	FOR NB2 := 1 TO NB_GROUP DO
		IF TBL_GROUP[NB2].NOM	= '' THEN
			IF NB2 < NB_GROUP THEN
				IF TBL_GROUP[NB2+1].NOM	<> '' THEN
					TBL_GROUP[NB2].NOM				:=	TBL_GROUP[NB2+1].NOM;
					TBL_GROUP[NB2].CONF_MACHINE	:=	TBL_GROUP[NB2+1].CONF_MACHINE;
					TBL_GROUP[NB2].FONCTION_SA		:=	TBL_GROUP[NB2+1].FONCTION_SA;
					TBL_GROUP[NB2].MAINTENANCE		:=	TBL_GROUP[NB2+1].MAINTENANCE;
					TBL_GROUP[NB2].PRODUCTION		:=	TBL_GROUP[NB2+1].PRODUCTION;
					TBL_GROUP[NB2].PROGRAMMATION	:=	TBL_GROUP[NB2+1].PROGRAMMATION;
					TBL_GROUP[NB2].SUPERVISEUR		:=	TBL_GROUP[NB2+1].SUPERVISEUR;
					TBL_GROUP[NB2].CONF_TRF			:=	TBL_GROUP[NB2+1].CONF_TRF;
					TBL_GROUP[NB2].MODIF_ENLIGNE	:=	TBL_GROUP[NB2+1].MODIF_ENLIGNE;
					TBL_GROUP[NB2].ARCHIVE_EV		:=	TBL_GROUP[NB2+1].ARCHIVE_EV;
					TBL_GROUP[NB2].DECONSIGNATION	:=	TBL_GROUP[NB2+1].DECONSIGNATION;
					TBL_GROUP[NB2+1].NOM				:=	'';
					TBL_GROUP[NB2+1].CONF_MACHINE	:=	FALSE;
					TBL_GROUP[NB2+1].FONCTION_SA	:=	FALSE;
					TBL_GROUP[NB2+1].MAINTENANCE	:=	FALSE;
					TBL_GROUP[NB2+1].PRODUCTION		:=	FALSE;
					TBL_GROUP[NB2+1].PROGRAMMATION	:=	FALSE;
					TBL_GROUP[NB2+1].SUPERVISEUR		:=	FALSE;
					TBL_GROUP[NB2+1].CONF_TRF			:=	FALSE;
					TBL_GROUP[NB2+1].MODIF_ENLIGNE		:=	FALSE;
					TBL_GROUP[NB2+1].ARCHIVE_EV			:=	FALSE;
					TBL_GROUP[NB2+1].DECONSIGNATION	:=	FALSE;
				END_IF
			END_IF
		END_IF;
	END_FOR;

	DD_ORG_GRP	:=	FALSE;
END_IF
(*================================================================================================*)


(****************************************************** 	Organisation des utlisateurs après suppression **********************************************)
IF DD_ORG_USER THEN
	FOR NB := 1 TO NB_USER DO
		IF  TBL_USER[NB].LOGIN = '' THEN
			IF NB < NB_USER THEN
				IF  TBL_USER[NB+1].LOGIN <> '' THEN
					TBL_USER[NB].LOGIN		:=	TBL_USER[NB+1].LOGIN;
					TBL_USER[NB].GROUPE	:=	TBL_USER[NB+1].GROUPE;
					TBL_USER[NB].NOM		:=	TBL_USER[NB+1].NOM;
					TBL_USER[NB].PRENOM	:=	TBL_USER[NB+1].PRENOM;
					TBL_USER[NB].PASS		:=	TBL_USER[NB+1].PASS;
					TBL_USER[NB+1].LOGIN		:=	'';
					TBL_USER[NB+1].GROUPE		:=	'';
					TBL_USER[NB+1].NOM			:=	'';
					TBL_USER[NB+1].PRENOM	:=	'';
					TBL_USER[NB+1].PASS		:=	'';
				END_IF
			END_IF
		END_IF
	END_FOR

	DD_ORG_USER	:=	FALSE;
END_IF
(*================================================================================================*)



(****************************************************** 	Autorisation modification nom du groupe ***************************************************)
TROUV:=FALSE;
FOR NB := 1 TO NB_GROUP DO
	IF nb <> LIGNE_GROUP THEN
		IF TBL_GROUP[NB].NOM = GROUP_TEMP.NOM THEN
			TROUV := TRUE;
		END_IF
	END_IF
END_FOR
FOR NB := 1 TO NB_USER DO
	IF TBL_USER[NB].GROUPE = TBL_GROUP[LIGNE_GROUP].NOM AND TBL_GROUP[LIGNE_GROUP].NOM <> GROUP_TEMP.NOM THEN
		TROUV		:=	TRUE;
	END_IF
END_FOR
IF TROUV THEN
	AUT_NOM_GRP	:=	FALSE;
ELSE
	AUT_NOM_GRP	:=	TRUE;
END_IF
(*================================================================================================*)



(****************************************************** 	Autorisation modification nom des utilisateurs ***************************************************)
TROUV:=FALSE;
FOR NB := 1 TO NB_USER DO
	IF nb <> LIGNE THEN
		IF TBL_USER[NB].LOGIN = USER_TEMP.LOGIN THEN
			TROUV := TRUE;
		END_IF
	END_IF
END_FOR
IF TROUV THEN
	AUT_NOM_USER	:=	FALSE;
ELSE
	AUT_NOM_USER	:=	TRUE;
END_IF
(*================================================================================================*)



(****************************************************** 	Autorisation création utilisateur ***************************************************)
IF USER_TEMP.LOGIN = '' OR USER_TEMP.PASS = '' OR USER_TEMP.PASS <> PASS_CONF OR USER_TEMP.LOGIN = 'ac' THEN
	AUT_NEW_USER	:=	FALSE;
ELSE
	AUT_NEW_USER	:=	TRUE;
END_IF
(*================================================================================================*)


(********************************************************** Gestion du logout automatique **************************************************)
IF OPT_LOGOUT THEN
	TPS_ECOUL.IN		:=	UTIL_EC AND NOT MANUFACTURER;
	TPS_ECOUL.PT	:=	TIM_LOGOUT;
	TPS_ECOUL();
	IF TPS_ECOUL.Q AND NOT MACHINE.STATE_Prod THEN
		DD_DELOG	:=	TRUE;
	END_IF
END_IF
(*=========================================================================================*)

(********************************************************** Autorisation utilisation logout auto **************************************************)
IF TIM_LOGOUT > T#10s THEN
	AUT_OPT_LOGOUT	:=	TRUE;
ELSE
	AUT_OPT_LOGOUT	:=	FALSE;
END_IF
(*=========================================================================================*)

END_FUNCTION_BLOCK

// ---- POUs/Programme/BLOCK_PRG_EFFLUVAGE.TcPOU
FUNCTION_BLOCK BLOCK_PRG_EFFLUVAGE
VAR
END_VAR
VAR_INPUT PERSISTENT
(* Entité*)
	IsAssembly:			 	BOOL;					(*entité de type fonction*)
	TagXml:					UINT;
	IdXml: 					STRING;
	IdParent: 				STRING;					(*MNEMO du pére*)
	MNEMO:					STRING;					(*MNEMO de cette entité *)
END_VAR
VAR_INPUT
END_VAR
VAR_OUTPUT
	STATE_AR:				BOOL;
	STATE_Def_IProc:		BOOL;		(*I_STANDARD -indique la présence d'un défaut entrainant l'arrêt du procédé*)
END_VAR

(* Parametre statique *)
(*General*)
IdParent			:= 	'';
MNEMO				:=	'EFFLUV';
IdXML				:=	'15';
TagXML				:=	0;


STATE_AR := TRUE;
STATE_Def_IProc := FALSE;

END_FUNCTION_BLOCK

// ---- POUs/Programme/BLOCK_PRG_EVAP.TcPOU
FUNCTION_BLOCK BLOCK_PRG_EVAP
VAR_INPUT
(*Quartz*)
	QZ1:				BLOCK_XTAL6; 	(*Tête Quartz*)
	XTC3:				BLOCK_XTC3;	(*Contrôleur de dépôt XTC3*)

(*Evenement*)
	EV_SHUTTER1_OPEN:	PRCDEF;		(*Evenement cache source 1 ouvert*)
	EV_SHUTTER1_CLOSE:	PRCDEF;		(*Evenement cache source 1 fermé*)

	EV_SHUTTER2_OPEN:	PRCDEF;		(*Evenement cache source 2 ouvert*)
	EV_SHUTTER2_CLOSE:	PRCDEF;		(*Evenement cache source 2 fermé*)

	EV_SHUTTER3_OPEN:	PRCDEF;		(*Evenement cache source 3 ouvert*)
	EV_SHUTTER3_CLOSE:	PRCDEF;		(*Evenement cache source 3 fermé*)

(*Entrées*)
	(*Creuset*)
	IN_CR11T		AT%I*:		BOOL;		(*Creuset en position 1*)
	IN_CR12T		AT%I*:		BOOL;		(*Creuset en position 2*)
	IN_CR13T		AT%I*:		BOOL;		(*Creuset en position 3*)
	IN_CR14T		AT%I*:		BOOL;		(*Creuset en position 4*)

	(*Balayage*)
	IN_SW_REM		AT%I*:		BOOL;		(*Balayage en mode remote*)
	IN_SW_RUN		AT%I*:		BOOL;		(*Balayage en marche*)
	IN_SW_RDY		AT%I*:		BOOL;		(*Balayage prêt*)

	VISU_STOP_ECO_MANU:			BOOL;
END_VAR
VAR_INPUT PERSISTENT
	(*Entité*)
	IsAssembly:		BOOL;			(*entité : ensemble*)
	IdXML:			STRING;			(*nom entité : identifiant pour recherche dans dico*)
	TagXML:			UINT;			(*nom entité : identifiant pour recherche dans dico*)
	IdParent:		STRING;			(*MNEMO de l'appelant*)
	MNEMO:			STRING;			(*MNEMO de l'entité*)

	CONF_QUARTZ_CC_SRCE:	ARRAY[0..4] OF BOOL;	(*Indique si un Quartz se trouve sous le cache source pour contrôle vitesse pendant phase de préfusion*)
	CONF_CHAUFFAGE:			BOOL; 	(*Indique s'il y a du chauffage*)
	CONF_IAD:				BOOL;	(*Indique s'il y a un IAD*)

	PRM_Seuil_Crystal_Life:			REAL;	(*Seuil d'alarme pour la vie des quartz*)
	PRM_Seuil_Crystal_Activity:		REAL;	(*Seuil d'alarme pour l'activité des quartz*)

	PRM_Forcage_Crucible:		BOOL;	(*Option de forçage du creuset en semi-auto*)
	PRM_Forcage_Cache_Source1:	BOOL;	(*Option de forçage du cache source 1 en semi-auto*)
	PRM_Forcage_Cache_Source2:	BOOL;	(*Option de forçage du cache source 2 en semi-auto*)
	PRM_Forcage_Cache_Source3:	BOOL;	(*Option de forçage du cache source 3 en semi-auto*)
	PRM_Forcage_Cache_Quartz:	BOOL;	(*Option de forçage du cache quartz en semi-auto*)

	PRM_Adresse_IP_XTC:			STRING(15) := '192.168.0.20'; (*Addresse IP de l'XTC affecté depuis l'IHM*)

	PRM_Mat_Source2:			STRING; (*Nom du matériau utilisé sur la source 2*)
	PRM_Mat_Source3:			STRING; (*Nom du matériau utilisé sur la source 3*)
END_VAR

VAR
	EVAPS1:			BLOCK_EVAP;
	EVAPS2:			BLOCK_EVAP;
	EVAPS3:			BLOCK_EVAP;
	CC11:			BLOCK_ACTUATOR;
	CC12:			BLOCK_ACTUATOR;
	CC13:			BLOCK_ACTUATOR;
	SOURCE1:		BLOCK_CANON_ST10;
	SOURCE2:		BLOCK_SOURCE_JOULE;
	SOURCE3:		BLOCK_SOURCE_JOULE;
	SWEEP1:			BLOCK_TELEMARK_CHEETAH_SWEEP;
	CRUCIBLE1:		BLOCK_IND_CR_396_TELEMARK;

	VAR_Idx:		INT;				(*Variable d'itération*)

	(*Variable Bidon*)
	VAR_NCR:				USINT;
	VAR_NBAL:				USINT;
	VAR_HT:					REAL;
END_VAR

VAR_OUTPUT
	STATE_AR:						BOOL;
	STATE_Def_IProc:   				BOOL;		(*Etat de défaut*)
	(*Caches*)
	OUT_OCC11			AT%Q*:		BOOL;		(*Ouverture cache source 1*)
	OUT_ICC11			AT%Q*:		BOOL;		(*Fermeture cache source 1*)
	OUT_OCC12			AT%Q*:		BOOL;		(*Ouverture cache source 2*)
	OUT_ICC12			AT%Q*:		BOOL;		(*Fermeture cache source 2*)
	OUT_OCC13			AT%Q*:		BOOL;		(*Ouverture cache source 3*)
	OUT_ICC13			AT%Q*:		BOOL;		(*Fermeture cache source 3*)
	(*Creuset*)
	OUT_CR11			AT%Q*:		BOOL;		(*Sélection du creuset 1*)
	OUT_CR12			AT%Q*:		BOOL;		(*Sélection du creuset 2*)
	OUT_CR13			AT%Q*:		BOOL;		(*Sélection du creuset 3*)
	OUT_CR14			AT%Q*:		BOOL;		(*Sélection du creuset 4*)
	OUT_CR_RMT			AT%Q*:		BOOL;		(*remote indexeur de creuset*)
	(*Sweep*)
	OUT_SWB1			AT%Q*:		BOOL;		(*Sélection programme de balayage bit 1*)
	OUT_SWB2			AT%Q*:		BOOL;		(*Sélection programme de balayage bit 2*)
	OUT_SWB3			AT%Q*:		BOOL;		(*Sélection programme de balayage bit 3*)
	OUT_SWB4			AT%Q*:		BOOL;		(*Sélection programme de balayage bit 4*)
	//OUT_SWITLK			AT%Q*:		BOOL;		(*Interlock module balayage*)
	OUT_SWP_ON			AT%Q*:		BOOL;		(*activation balayage*)
	OUT_SW_RMT			AT%Q*:		BOOL;		(*remote module de balayage*)
	(*Effet joule*)
	OUT_MEJ1			AT%Q*:		BOOL;
	OUT_MEJ2			AT%Q*:		BOOL;
	OUT_QEJ1			AT%Q*:		INT;
	OUT_QEJ2			AT%Q*:		INT;
	
	(*Divers*)
	OUT_MEG1			AT%Q*:		BOOL;		(*Sécurité vide canon pour mise en puissance canons + ECO-MODE*)
	OUT_MPR230			AT%Q*:		BOOL;		(*230V Module Balayage + Module Indexage + XTC ECO-MODE*)
	ECO_MODE:						BOOL;

	O_END_PROCESS_PFIXE:			BOOL;		(**)
END_VAR

VAR
	TIMER_ECO_MODE:					TOF;
END_VAR

(*General*)
IdParent					:=	MACHINE.MNEMO;
MNEMO						:=	CONCAT(IdParent,'_EVAP');
IdXML						:=	'17';
TagXML						:=	0;

(*XTC3*)
XTC3.MNEMO					:=	'XTC3';
XTC3.IdXML					:=	'19';
XTC3.TagXML					:=	1;

(*Quartz*)
QZ1.MNEMO					:=	'QZ1';
QZ1.IdParent				:=	MNEMO;

(*Source1*)
SOURCE1.IdParent			:=	MNEMO;
SOURCE1.MNEMO				:=	'Canon e-';
SOURCE1.IdXML				:=	'16';
SOURCE1.TagXML 				:= 	3;

(*Source2*)
SOURCE2.IdParent			:=	MNEMO;
SOURCE2.MNEMO				:=	'Source J-Gauche';
SOURCE2.IdXML				:=	'16';
SOURCE2.TagXML				:=	4;

(*Source3*)
SOURCE3.IdParent			:=	MNEMO;
SOURCE3.MNEMO				:=	'Source J-Droite';
SOURCE3.IdXML				:=	'16';
SOURCE3.TagXML				:=	5;

(*Balayage*)
SWEEP1.IdParent				:=	SOURCE1.MNEMO;
SWEEP1.MNEMO				:=	'SWP1';
SWEEP1.IdXML				:=	'16';
SWEEP1.TagXML				:=	8;

(*Indexeur*)
CRUCIBLE1.IdParent 			:=	SOURCE1.MNEMO;
CRUCIBLE1.MNEMO 			:=	'INDCR1';
CRUCIBLE1.IdXML				:=	'16';
CRUCIBLE1.TagXML 			:=  7;

CRUCIBLE1.CONF_NCR			:= 	4;			(*Nombre de creuset de l'indexeur*)

(*Cache CC11*)
CC11.CONF_Tim_Valid_Off			:=	T#0ms;
CC11.CONF_Tim_Valid_On			:=	T#0ms;
CC11.DEF_Off.DELAY				:=	T#10s;
CC11.DEF_On.DELAY				:=	T#10s;
CC11.DEF_Sensor.DELAY			:=	T#10s;
CC11.CONF_DI_Off				:=	FALSE;
CC11.CONF_DI_On					:=	FALSE;
CC11.CONF_No_Safety_Auto		:=	TRUE;
CC11.CONF_Type_Actuator			:=	0;
CC11.MNEMO						:=	'Canon e-';
CC11.CONF_EN_On					:=	0;
CC11.CONF_No_Safety_Auto		:=	FALSE;
CC11.IdXML						:=	'4';
CC11.TagXML						:=	1;
CC11.IdParent					:=	Source1.MNEMO;
CC11.DEF_Off_auto.IdXML			:=	'3';
CC11.DEF_Off_auto.TagXML		:=	11;
CC11.DEF_Off_Imposs.IdXML		:=	'3';
CC11.DEF_Off_Imposs.TagXML		:=	9;
CC11.DEF_On_Imposs.IdXML		:=	'3';
CC11.DEF_On_Imposs.TagXML		:=	6;
CC11.DEF_Off.IdXML				:=	'3';
CC11.DEF_Off.TagXML 			:=	4;
CC11.DEF_On.IdXML				:=	'3';
CC11.DEF_On.TagXML 				:=	2;
CC11.DEF_Sensor.IdXML			:=	'3';
CC11.DEF_Sensor.TagXML 			:=	13;

(*Cache CC12*)
CC12.CONF_Tim_Valid_Off			:=	T#0ms;
CC12.CONF_Tim_Valid_On			:=	T#0ms;
CC12.DEF_Off.DELAY				:=	T#10s;
CC12.DEF_On.DELAY				:=	T#10s;
CC12.DEF_Sensor.DELAY			:=	T#10s;
CC12.CONF_DI_Off				:=	FALSE;
CC12.CONF_DI_On					:=	FALSE;
CC12.CONF_No_Safety_Auto		:=	TRUE;
CC12.CONF_Type_Actuator			:=	0;
CC12.MNEMO						:=	'SJ-Gauche';
CC12.CONF_EN_On					:=	0;
CC12.CONF_No_Safety_Auto		:=	FALSE;
CC12.IdXML						:=	'4';
CC12.TagXML						:=	1;
CC12.IdParent					:=	Source2.MNEMO;
CC12.DEF_Off_auto.IdXML			:=	'3';
CC12.DEF_Off_auto.TagXML		:=	11;
CC12.DEF_Off_Imposs.IdXML		:=	'3';
CC12.DEF_Off_Imposs.TagXML		:=	9;
CC12.DEF_On_Imposs.IdXML		:=	'3';
CC12.DEF_On_Imposs.TagXML		:=	6;
CC12.DEF_Off.IdXML				:=	'3';
CC12.DEF_Off.TagXML 			:=	4;
CC12.DEF_On.IdXML				:=	'3';
CC12.DEF_On.TagXML 				:=	2;
CC12.DEF_Sensor.IdXML			:=	'3';
CC12.DEF_Sensor.TagXML 			:=	13;

(*Cache CC13*)
CC13.CONF_Tim_Valid_Off			:=	T#0ms;
CC13.CONF_Tim_Valid_On			:=	T#0ms;
CC13.DEF_Off.DELAY				:=	T#10s;
CC13.DEF_On.DELAY				:=	T#10s;
CC13.DEF_Sensor.DELAY			:=	T#10s;
CC13.CONF_DI_Off				:=	FALSE;
CC13.CONF_DI_On					:=	FALSE;
CC13.CONF_No_Safety_Auto		:=	TRUE;
CC13.CONF_Type_Actuator			:=	0;
CC13.MNEMO						:=	'SJ-Droite';
CC13.CONF_EN_On					:=	0;
CC13.CONF_No_Safety_Auto		:=	FALSE;
CC13.IdXML						:=	'4';
CC13.TagXML						:=	1;
CC13.IdParent					:=	Source3.MNEMO;
CC13.DEF_Off_auto.IdXML			:=	'3';
CC13.DEF_Off_auto.TagXML		:=	11;
CC13.DEF_Off_Imposs.IdXML		:=	'3';
CC13.DEF_Off_Imposs.TagXML		:=	9;
CC13.DEF_On_Imposs.IdXML		:=	'3';
CC13.DEF_On_Imposs.TagXML		:=	6;
CC13.DEF_Off.IdXML				:=	'3';
CC13.DEF_Off.TagXML 			:=	4;
CC13.DEF_On.IdXML				:=	'3';
CC13.DEF_On.TagXML 				:=	2;
CC13.DEF_Sensor.IdXML			:=	'3';
CC13.DEF_Sensor.TagXML 			:=	13;

EVAPS1.IdXML 				:=	'17';
EVAPS1.TagXML				:=	1;
EVAPS1.CONF_No_Sweep		:=	FALSE;
EVAPS1.DEF_Pmax.DELAY		:=	T#10S;
EVAPS1.DEF_Pmin.DELAY		:=	T#10s;

EVAPS2.IdXML				:=	'17';
EVAPS2.TagXML				:=	2;
EVAPS2.CONF_No_Sweep		:=	TRUE;
EVAPS2.DEF_Pmax.DELAY		:=	T#10S;
EVAPS2.DEF_Pmin.DELAY		:=	T#10s;

EVAPS3.IdXML				:=	'17';
EVAPS3.TagXML				:=	3;
EVAPS3.CONF_No_Sweep		:=	TRUE;
EVAPS3.DEF_Pmax.DELAY		:=	T#10S;
EVAPS3.DEF_Pmin.DELAY		:=	T#10s;


EV_SHUTTER1_OPEN.IdXML			:=	'14';
EV_SHUTTER1_OPEN.TagXML			:=	20;
EV_SHUTTER1_OPEN.Groupe			:=	3;

EV_SHUTTER1_CLOSE.IdXML			:=	'14';
EV_SHUTTER1_CLOSE.TagXML		:=	21;
EV_SHUTTER1_CLOSE.Groupe		:=	3;

EV_SHUTTER2_OPEN.IdXML			:=	'14';
EV_SHUTTER2_OPEN.TagXML			:=	24;
EV_SHUTTER2_OPEN.Groupe			:=	3;

EV_SHUTTER2_CLOSE.IdXML			:=	'14';
EV_SHUTTER2_CLOSE.TagXML		:=	25;
EV_SHUTTER2_CLOSE.Groupe		:=	3;

EV_SHUTTER3_OPEN.IdXML			:=	'14';
EV_SHUTTER3_OPEN.TagXML			:=	26;
EV_SHUTTER3_OPEN.Groupe			:=	3;

EV_SHUTTER3_CLOSE.IdXML			:=	'14';
EV_SHUTTER3_CLOSE.TagXML		:=	27;
EV_SHUTTER3_CLOSE.Groupe		:=	3;


CONF_CHAUFFAGE:= FALSE;
CONF_IAD:=FALSE;

CONF_QUARTZ_CC_SRCE[0]:= FALSE;
CONF_QUARTZ_CC_SRCE[1]:= FALSE;
CONF_QUARTZ_CC_SRCE[2]:= FALSE;
CONF_QUARTZ_CC_SRCE[3]:= FALSE;
CONF_QUARTZ_CC_SRCE[4]:= FALSE;


(*mode de controle des fonctions*)
IF MACHINE.RQ_Ctrl_Ihm THEN
	QZ1.CTRL_PLC := FALSE;
ELSIF MACHINE.RQ_Ctrl_Plc THEN
	QZ1.CTRL_PLC := TRUE;
END_IF

(*Configuration Adresse IP XTC*)
XTC3.CONF_sRemoteHost:= PRM_Adresse_IP_XTC;
XTC3.CONF_nRemotePort := 2101;


(*Evenement ouverture cache source 1*)
EV_SHUTTER1_OPEN.CONDITION	:= MACHINE.STATE_Prod AND CC11.STATE_On;
EV_SHUTTER1_OPEN();
(*Evenement fermeture cache source 1*)
EV_SHUTTER1_CLOSE.CONDITION:= MACHINE.STATE_Prod AND CC11.STATE_Off;
EV_SHUTTER1_CLOSE();

(*Evenement ouverture cache source 2*)
EV_SHUTTER2_OPEN.CONDITION	:= MACHINE.STATE_Prod AND CC12.STATE_On;
EV_SHUTTER2_OPEN();
(*Evenement fermeture cache source 2*)
EV_SHUTTER2_CLOSE.CONDITION:= MACHINE.STATE_Prod AND CC12.STATE_Off;
EV_SHUTTER2_CLOSE();

(*Evenement ouverture cache source 3*)
EV_SHUTTER3_OPEN.CONDITION	:= MACHINE.STATE_Prod AND CC13.STATE_On;
EV_SHUTTER3_OPEN();
(*Evenement fermeture cache source 3*)
EV_SHUTTER3_CLOSE.CONDITION:= MACHINE.STATE_Prod AND CC13.STATE_Off;
EV_SHUTTER3_CLOSE();


(*Reset des ordres de forçage*)
IF MACHINE.RQ_Start_Prod OR MACHINE.STATE_Off OR MACHINE.STATE_Manu THEN
	PRM_Forcage_Crucible 		:= 	FALSE;
	PRM_Forcage_Cache_Source1	:= 	FALSE;
	PRM_Forcage_Cache_Source2	:=	FALSE;
	PRM_Forcage_Cache_Source3  	:=	FALSE;
	PRM_Forcage_Cache_Quartz	:=	FALSE;
END_IF
IF CRUCIBLE1.DEF_POSITIONNEMENT.DEF THEN
	PRM_Forcage_Crucible		:= FALSE;
END_IF
IF CC11.DEF_Off_auto.DEF THEN
	PRM_Forcage_Cache_Source1:= FALSE;
END_IF
IF CC12.DEF_Off_auto.DEF	THEN
	PRM_Forcage_Cache_Source2:= FALSE;
END_IF
IF CC13.DEF_Off_auto.DEF	THEN
	PRM_Forcage_Cache_Source3:= FALSE;
END_IF


(******************* SOURCE 1 **********************)

SOURCE1.HV.EN_Off_EXT := TRUE;
SOURCE1.HV.EN_On_EXT := (SWEEP1.STATE_REM AND SWEEP1.STATE_ON);

SOURCE1(
	DOOR:= PRG_POMPAGE.DOOR,
	VAC:= (PRG_POMPAGE.VAC AND PRG_POMPAGE.M11.STATE_Seuil[13] AND NOT PRG_POMPAGE.POMPAGE.VS11.STATE_Off),
	WATER:= PRG_SERVITUDES.WATER[4] AND PRG_SERVITUDES.WATER[5],	(*Refroidissement canon à électrons*)
	MANUAL:= MACHINE.STATE_Manu,
	I_CR_OK:= CRUCIBLE1.STATE_POS_OK,
	RESET:= MACHINE.STATE_Off,
	I_COURANT:= EVAPS1.OUT_Power,
	CO_HV:= EVAPS1.RQ_marche_HT,
	CO_SRC:=EVAPS1.RQ_marche_FIL ,);

SWEEP1(
	MANUAL:= MACHINE.STATE_Manu,
	RESET:= MACHINE.STATE_Off,
	DOOR:= PRG_POMPAGE.DOOR,
	CO_Remote:= MACHINE.STATE_Auto,
	CO_balayage:= MACHINE.STATE_Auto AND EVAPS1.RQ_marche_SWEEP,
	I_SW_RUN:= IN_SW_RUN,
	I_SW_RDY:= IN_SW_RDY,
	OUT_SWB1 => OUT_SWB1,
	OUT_SWB2 => OUT_SWB2,
	OUT_SWB3 => OUT_SWB3,
	OUT_SWB4 => OUT_SWB4,
	OUT_SWP_ON => OUT_SWP_ON,
	OUT_RMT	=> OUT_SW_RMT);

CRUCIBLE1(
	MANUAL:= MACHINE.STATE_Manu,
	RESET:= MACHINE.STATE_Off,
	CO_Change:= EVAPS1.RQ_Switch_Crucible OR PRM_Forcage_Crucible,
	I_FIL_ON:= SOURCE1.STATE_SRC_ON,
	IN_POWER:= EVAPS1.OUT_Power,
	IN_POS1:= IN_CR11T,
	IN_POS2:= IN_CR12T,
	IN_POS3:= IN_CR13T,
	IN_POS4:= IN_CR14T,
	OUT_SEL1=> OUT_CR11,
	OUT_SEL2=> OUT_CR12,
	OUT_SEL3=> OUT_CR13,
	OUT_SEL4=> OUT_CR14);

CC11(
	RESET:= MACHINE.STATE_Off ,
	MANUAL:=MACHINE.STATE_Manu,
	IN_OFF:= ,
	IN_ON:= ,
	CO_On:= EVAPS1.RQ_Ouv_Cache_source OR PRM_Forcage_Cache_Source1,
	CO_Off:= NOT EVAPS1.RQ_Ouv_Cache_source AND NOT PRM_Forcage_Cache_Source1 AND NOT MACHINE.STATE_Manu AND NOT MACHINE.STATE_Off,
	EN_On_INT:= TRUE,
	EN_Off_INT:= TRUE,
	EN_On_EXT:=TRUE,
	EN_Off_EXT:= TRUE,
	OUT_On=> OUT_OCC11,
	OUT_Off=> OUT_ICC11,);
	

(******************* SOURCE 2 **********************)

SOURCE2.EJ.EN_Off_EXT	:=	TRUE;
SOURCE2.EJ.EN_On_EXT	:=	NOT SOURCE3.OUT_MEJ;

SOURCE2(
	DOOR:=					PRG_POMPAGE.DOOR,
	VAC:=					PRG_POMPAGE.VAC AND NOT PRG_POMPAGE.POMPAGE.VS11.STATE_Off,
	WATER:=					PRG_SERVITUDES.WATER[2],					(*Refroidissement Source Joule n°1*)
	MANUAL:=				MACHINE.STATE_Manu,
	I_CR_OK:=				TRUE,										(*Positionnement du creuset ok*)
	RESET:=					MACHINE.STATE_Off,
	I_POWER:=				EVAPS2.OUT_Power,
	CO_SRC:=				EVAPS2.RQ_marche_HT, );

CC12(
	RESET:= MACHINE.STATE_Off ,
	MANUAL:=MACHINE.STATE_Manu,
	IN_OFF:= ,
	IN_ON:= ,
	CO_On:= EVAPS2.RQ_Ouv_Cache_source OR PRM_Forcage_Cache_Source2,
	CO_Off:= NOT EVAPS2.RQ_Ouv_Cache_source AND NOT PRM_Forcage_Cache_Source2 AND NOT MACHINE.STATE_Manu AND NOT MACHINE.STATE_Off,
	EN_On_INT:= TRUE,
	EN_Off_INT:= TRUE,
	EN_On_EXT:=TRUE,
	EN_Off_EXT:= TRUE,
	OUT_On=> OUT_OCC12,
	OUT_Off=> OUT_ICC12);

(******************* SOURCE 3 **********************)

SOURCE3.EJ.EN_Off_EXT	:=	TRUE;
SOURCE3.EJ.EN_On_EXT	:=	NOT SOURCE2.OUT_MEJ;

SOURCE3(
	DOOR:=					PRG_POMPAGE.DOOR,
	VAC:=					PRG_POMPAGE.VAC AND NOT PRG_POMPAGE.POMPAGE.VS11.STATE_Off,
	WATER:=					PRG_SERVITUDES.WATER[3],					(*Refroidissement Source Joule n°2*)
	MANUAL:=				MACHINE.STATE_Manu,
	I_CR_OK:=				TRUE,										(*Positionnement du creuset ok*)
	RESET:=					MACHINE.STATE_Off,
	I_POWER:=				EVAPS3.OUT_Power,
	CO_SRC:=				EVAPS3.RQ_marche_HT,	);

	
CC13(
	RESET:= MACHINE.STATE_Off ,
	MANUAL:= MACHINE.STATE_Manu,
	IN_OFF:= ,
	IN_ON:= ,
	CO_On:= EVAPS3.RQ_Ouv_Cache_source OR PRM_Forcage_Cache_Source3,
	CO_Off:= NOT EVAPS3.RQ_Ouv_Cache_source AND NOT PRM_Forcage_Cache_Source3 AND NOT MACHINE.STATE_Manu AND NOT MACHINE.STATE_Off,
	EN_On_INT:= TRUE,
	EN_Off_INT:= TRUE,
	EN_On_EXT:=TRUE,
	EN_Off_EXT:= TRUE,
	OUT_On=> OUT_OCC13,
	OUT_Off=> OUT_ICC13,);
	
(******************* QUARTZ **********************)

(*Quartz QZ1*)
IF MACHINE.STATE_Prod THEN
	IF MAIN.STEP_EMPILEMENT.PRM_UTIL_SOURCE1 THEN
		QZ1.PRM_CONS_POSITION_QZ:= EVAPS1.OUT_Cons_Pos_Qz;
	END_IF
	IF MAIN.STEP_EMPILEMENT.PRM_UTIL_SOURCE2 THEN
		QZ1.PRM_CONS_POSITION_QZ:= EVAPS2.OUT_Cons_Pos_Qz;
	END_IF
	IF MAIN.STEP_EMPILEMENT.PRM_UTIL_SOURCE3 THEN
		QZ1.PRM_CONS_POSITION_QZ:= EVAPS3.OUT_Cons_Pos_Qz;
	END_IF
	IF MODE_QUARTZ_PROD.RQ_Pos_Quartz THEN
		QZ1.PRM_CONS_POSITION_QZ:= MODE_QUARTZ_PROD.OUT_Quartz;
	END_IF
END_IF

QZ1.OP_Scan_Quartz.ENABLE_EXT :=  NOT XTC3.STATE_NOK AND NOT MACHINE.STATE_Prod;
QZ1.OP_Positionnement.ENABLE_EXT := NOT XTC3.STATE_NOK;

QZ1.OP_Positionnement.ON_PLC:= EVAPS1.RQ_Switch_Crystal OR EVAPS2.RQ_Switch_Crystal OR EVAPS3.RQ_Switch_Crystal OR MODE_QUARTZ_PROD.RQ_Pos_Quartz;

QZ1	(
	RESET:= 					MACHINE.STATE_Off ,
	MANUAL:=					MACHINE.STATE_Manu ,
	CO_SWITCH_CRYSTAL:=			XTC3.OUT_CACHE_QUARTZ,
	IN_QF:=						XTC3.STATE_Sensor_Fail,
	IN_RATE:=					XTC3.STATE_Rate,
	IN_FREQ:= 					XTC3.STATE_Frequency,
	IN_THICKNESS:= 				XTC3.STATE_Thickness,
	IN_LIFE:= 					XTC3.STATE_Crystal_Life,
	IN_ACTIVITY:=				,
	PRM_Seuil_Life:=			PRM_Seuil_Crystal_Life,
	PRM_Seuil_Activity:=		,
	RQ_SWITCH_CRYSTAL=>			XTC3.CO_Switch_Crystal,
	);

(******************* PILOTAGE DES QUARTZ **********************)

IF MODE_QUARTZ_PROD.STATE_Mode THEN
	EVAPS1.PRM_CRYSTAL_POSITION		:=	MODE_QUARTZ_PROD.OUT_Quartz;
	EVAPS2.PRM_CRYSTAL_POSITION		:=	MODE_QUARTZ_PROD.OUT_Quartz;
	EVAPS3.PRM_CRYSTAL_POSITION		:=	MODE_QUARTZ_PROD.OUT_Quartz;
END_IF

(******************* EVAPORATION  S1 **********************)

EVAPS1.OP_Marche.ENABLE_EXT := TRUE;
EVAPS1.OP_Stop.ENABLE_EXT := TRUE;
(*Demande marche source par bloc empilement*)
EVAPS1.OP_Marche.ON_PLC := MAIN.STEP_EMPILEMENT.RQ_PREP_S1;
EVAPS1.OP_Stop.ON_PLC := MAIN.STEP_EMPILEMENT.RQ_STOP_EVAP_S1 OR INIT_MACHINE.RQ_STOP_EVAP ;

EVAPS1(
	RESET:=MACHINE.STATE_Off ,
	MANUAL:= MACHINE.STATE_Manu ,
	I_END_DEPOSITION:= NOT MAIN.STEP_EMPILEMENT.RQ_EVAP_S1 OR INIT_MACHINE.RQ_STOP_EVAP,
	I_EVAP_ON:= MAIN.STEP_EMPILEMENT.RQ_EVAP_S1,
	I_DEF_QZ_CTRL_RATE:= XTC3.STATE_Sensor_Fail,
	I_TIME_POWER:= XTC3.I_Time_Power,
	CO_FIN_ETAPE:= MAIN.STEP_EMPILEMENT.RQ_NEXT_LAYER,
	I_THICKNESS:= XTC3.STATE_Thickness,		(*Epaisseur global déposé*)
	I_cache_ouvert:= CC11.STATE_On,
	I_cache_ferme:= CC11.STATE_Off,
	I_ref_source_ok:= PRG_SERVITUDES.WATER[4] AND PRG_SERVITUDES.WATER[5],	(*Refroidissement Canon*)
	I_ref_mesure_ok:= PRG_SERVITUDES.WATER[1],	(*Refroidissement Quartz*)
	I_retour_pos_creuset_ok:= CRUCIBLE1.STATE_POS_OK ,
	I_HT_ON:=SOURCE1.STATE_HV_ON,
	I_HT_OFF:= NOT SOURCE1.STATE_HV_ON,
	I_FIL_ON:= SOURCE1.STATE_SRC_ON,
	I_FIL_OFF:= NOT SOURCE1.STATE_SRC_ON,
	I_SWEEP_ON := SWEEP1.STATE_ON,
	I_Power:= XTC3.STATE_Power,
	I_SWITCH_XTAL_OK:= QZ1.STATE_SELECT_QZ_OK,
	I_OUV_CACHE_SOURCE:= XTC3.OUT_CACHE_SRCE,
	PRM_Quartz_Cache_Source:= CONF_QUARTZ_CC_SRCE[0],
	PRM_THICKNESS := MAIN.STEP_EMPILEMENT.PRM_EPAISSEUR,
	PRM_MULTI_QUARTZ:= TRUE,
	CONS_NCR:= CRUCIBLE1.PRM_NCR,
	CONS_NBAL:= SWEEP1.PRM_NbBal,
	CONS_HT := SOURCE1.I_TENSION,
	STATE_Segment=> ,
	STATE_TEMPS_PREPARATION=> ,
	STATE_TEMPS_CLOTURE=> ,
	STATE_TEMPS_DEPOT=> ,
	STATE_TEMPS_RESTANT_PREP=> ,
	STATE_TEMPS_RESTANT_CLOT=> ,
	STATE_TEMPS_RESTANT_DEPOT=> ,
	OUT_Power=> ,
	RQ_ouv_cache_IAD=> ,
	RQ_Ref_source=> ,
	RQ_Ref_mesure=> ,
	RQ_Ouv_Cache_source=> ,
	RQ_marche_HT=> ,
	RQ_marche_FIL=> ,
	STATE_PREP_OK=> ,
	STATE_EVAP=> ,
	STATE_CLOT_OK=> ,
	STATE_AR=> );


(******************* EVAPORATION  S2 **********************)

EVAPS2.OP_Marche.ENABLE_EXT := 		TRUE;
EVAPS2.OP_Stop.ENABLE_EXT := 		TRUE;
(*Demande marche source par bloc empilement*)
EVAPS2.OP_Marche.ON_PLC :=			MAIN.STEP_EMPILEMENT.RQ_PREP_S2;
EVAPS2.OP_Stop.ON_PLC := 			MAIN.STEP_EMPILEMENT.RQ_STOP_EVAP_S2 OR INIT_MACHINE.RQ_STOP_EVAP;

(*recopie*)
EVAPS2.PRM_TPS_MIN_SURV_DEPOT	:=	EVAPS1.PRM_TPS_MIN_SURV_DEPOT;
EVAPS2.PRM_FACTEUR_TEMPS_DEPOT	:=	EVAPS1.PRM_FACTEUR_TEMPS_DEPOT;	

EVAPS2(
	RESET:=						MACHINE.STATE_Off,
	MANUAL:= 					MACHINE.STATE_Manu,
	I_END_DEPOSITION:= 			NOT MAIN.STEP_EMPILEMENT.RQ_EVAP_S2 OR INIT_MACHINE.RQ_STOP_EVAP,
	I_EVAP_ON:= 				MAIN.STEP_EMPILEMENT.RQ_EVAP_S2,
	I_DEF_QZ_CTRL_RATE:= 		XTC3.STATE_Sensor_Fail ,
	I_TIME_POWER:= 				XTC3.I_Time_Power,
	CO_FIN_ETAPE:= 				MAIN.STEP_EMPILEMENT.RQ_NEXT_LAYER ,
	I_THICKNESS:= 				XTC3.STATE_Thickness ,				(*Epaisseur global déposé*)
	I_cache_ouvert:= 			CC12.STATE_On ,
	I_cache_ferme:= 			CC12.STATE_Off ,
	I_ref_source_ok:= 			PRG_SERVITUDES.WATER[2],			(*Refroidissement Source Joule*)
	I_ref_mesure_ok:= 			PRG_SERVITUDES.WATER[1],			(*Refroidissement Quartz*)
	I_retour_pos_creuset_ok:= 	TRUE ,
	I_HT_ON:=  					SOURCE2.STATE_EJ_ON ,
	I_HT_OFF:= 					NOT SOURCE2.STATE_EJ_ON ,
	I_FIL_ON:= 					TRUE ,
	I_FIL_OFF:= 				TRUE ,
	I_Power:= 					XTC3.STATE_Power ,
	I_SWITCH_XTAL_OK:= 			QZ1.STATE_SELECT_QZ_OK,
	I_OUV_CACHE_SOURCE:= 		XTC3.OUT_CACHE_SRCE,
	PRM_Quartz_Cache_Source:= 	CONF_QUARTZ_CC_SRCE[0],
	PRM_THICKNESS := 			MAIN.STEP_EMPILEMENT.PRM_EPAISSEUR,
	PRM_MULTI_QUARTZ:= 			TRUE,
	PRM_HT:= 					10.0,
	CONS_NCR:= 					VAR_NCR ,
	CONS_NBAL:=					VAR_NBAL ,
	CONS_HT := 					VAR_HT ,
	);


(******************* EVAPORATION  S3 **********************)

EVAPS3.OP_Marche.ENABLE_EXT := 		TRUE;
EVAPS3.OP_Stop.ENABLE_EXT := 		TRUE;
(*Demande marche source par bloc empilement*)
EVAPS3.OP_Marche.ON_PLC :=			MAIN.STEP_EMPILEMENT.RQ_PREP_S3;
EVAPS3.OP_Stop.ON_PLC := 			MAIN.STEP_EMPILEMENT.RQ_STOP_EVAP_S3 OR INIT_MACHINE.RQ_STOP_EVAP;

(*recopie*)
EVAPS3.PRM_TPS_MIN_SURV_DEPOT	:=	EVAPS1.PRM_TPS_MIN_SURV_DEPOT;
EVAPS3.PRM_FACTEUR_TEMPS_DEPOT	:=	EVAPS1.PRM_FACTEUR_TEMPS_DEPOT;	

EVAPS3(
	RESET:=						MACHINE.STATE_Off,
	MANUAL:= 					MACHINE.STATE_Manu,
	I_END_DEPOSITION:= 			NOT MAIN.STEP_EMPILEMENT.RQ_EVAP_S3 OR INIT_MACHINE.RQ_STOP_EVAP,
	I_EVAP_ON:= 				MAIN.STEP_EMPILEMENT.RQ_EVAP_S3,
	I_DEF_QZ_CTRL_RATE:= 		XTC3.STATE_Sensor_Fail ,
	I_TIME_POWER:= 				XTC3.I_Time_Power,
	CO_FIN_ETAPE:= 				MAIN.STEP_EMPILEMENT.RQ_NEXT_LAYER ,
	I_THICKNESS:= 				XTC3.STATE_Thickness ,				(*Epaisseur global déposé*)
	I_cache_ouvert:= 			CC13.STATE_On ,
	I_cache_ferme:= 			CC13.STATE_Off ,
	I_ref_source_ok:= 			PRG_SERVITUDES.WATER[3],			(*Refroidissement Source Joule*)
	I_ref_mesure_ok:= 			PRG_SERVITUDES.WATER[1],			(*Refroidissement Quartz*)
	I_retour_pos_creuset_ok:= 	TRUE ,
	I_HT_ON:=  					SOURCE3.STATE_EJ_ON ,
	I_HT_OFF:= 					NOT SOURCE3.STATE_EJ_ON ,
	I_FIL_ON:= 					TRUE ,
	I_FIL_OFF:= 				TRUE ,
	I_Power:= 					XTC3.STATE_Power ,
	I_SWITCH_XTAL_OK:= 			QZ1.STATE_SELECT_QZ_OK,
	I_OUV_CACHE_SOURCE:= 		XTC3.OUT_CACHE_SRCE,
	PRM_Quartz_Cache_Source:= 	CONF_QUARTZ_CC_SRCE[0],
	PRM_THICKNESS := 			MAIN.STEP_EMPILEMENT.PRM_EPAISSEUR,
	PRM_MULTI_QUARTZ:= 			TRUE,
	PRM_HT:= 					10.0,
	CONS_NCR:= 					VAR_NCR ,
	CONS_NBAL:=					VAR_NBAL ,
	CONS_HT := 					VAR_HT ,
	);


(**********Contrôleur de dépôt XTC3***********)
(*transmission consignes depuis source utilisée*)
IF MAIN.STEP_EMPILEMENT.PRM_UTIL_SOURCE1 THEN
	XTC3.I_Soak_Power_2		:=	EVAPS1.PRM_SOAK2_POWER;
	XTC3.I_Deposition_Rate	:=	EVAPS1.PRM_Rate;
	XTC3.I_Thick_SP			:=	EVAPS1.PRM_Thick_SP;
	XTC3.I_New_Rate			:=	EVAPS1.PRM_New_Rate;
	XTC3.I_Rate_Ramp_Time	:=	EVAPS1.PRM_Rate_Ramp_Time;
	XTC3.I_Stab_Single		:=	EVAPS1.PRM_Stability_Single;
	XTC3.I_Stab_Total		:=	EVAPS1.PRM_Stability_Total;
	XTC3.I_Quality_Percent	:=	EVAPS1.PRM_Quality_Percent;
	XTC3.I_Quality_Counts	:=	EVAPS1.PRM_Quality_Counts;
	XTC3.I_PID_Gain			:=	EVAPS1.PRM_GAIN;
	XTC3.I_PID_Ti			:=	EVAPS1.PRM_INTEGRAL;
	XTC3.I_PID_Td			:=	EVAPS1.PRM_DERIVEE;
	XTC3.I_Max_Power		:=	EVAPS1.PRM_PMAX;
	IF EVAPS1.PRM_Quartz_Cache_Source AND EVAPS1.PRM_SHUTTER_Option THEN
		IF EVAPS1.PRM_CTRL_DELAY_TIME = 0 THEN
			XTC3.I_Delay_Option		:=	1; (*shutter*)
		ELSE
			XTC3.I_Delay_Option		:=	3; (*both*)
			XTC3.I_Ctrl_Delay_Time	:=	EVAPS1.PRM_CTRL_DELAY_TIME;
		END_IF
		(*
		XTC3.I_Transfer_Sensor		:=	1;
		XTC3.I_Transfer_Tool			:=	EVAPS1.PRM_Transfer_Tooling;	(*Pas de 2eme sensor sous cache *)
		*)
	ELSE
		IF EVAPS1.PRM_CTRL_DELAY_TIME = 0 THEN
			XTC3.I_Delay_Option		:=	0; (*none*)
		ELSE
			XTC3.I_Delay_Option		:=	2; (*controle*)
			XTC3.I_Ctrl_Delay_Time	:=	EVAPS1.PRM_CTRL_DELAY_TIME;
		END_IF
		(*
		XTC3.I_Transfer_Sensor		:=	0;								(*Pas de 2eme sensor sous cache*)
		*)
	END_IF
END_IF

IF MAIN.STEP_EMPILEMENT.PRM_UTIL_SOURCE2 THEN
	XTC3.I_Soak_Power_2		:=	EVAPS2.PRM_SOAK2_POWER;
	XTC3.I_Deposition_Rate	:=	EVAPS2.PRM_Rate;
	XTC3.I_Thick_SP			:=	EVAPS2.PRM_Thick_SP;
	XTC3.I_New_Rate			:=	EVAPS2.PRM_New_Rate;
	XTC3.I_Rate_Ramp_Time	:=	EVAPS2.PRM_Rate_Ramp_Time;
	XTC3.I_Stab_Single		:=	EVAPS2.PRM_Stability_Single;
	XTC3.I_Stab_Total		:=	EVAPS2.PRM_Stability_Total;
	XTC3.I_Quality_Percent	:=	EVAPS2.PRM_Quality_Percent;
	XTC3.I_Quality_Counts	:=	EVAPS2.PRM_Quality_Counts;
	XTC3.I_PID_Gain			:=	EVAPS2.PRM_GAIN;
	XTC3.I_PID_Ti			:=	EVAPS2.PRM_INTEGRAL;
	XTC3.I_PID_Td			:=	EVAPS2.PRM_DERIVEE;
	XTC3.I_Max_Power		:=	EVAPS2.PRM_PMAX;
	IF EVAPS2.PRM_Quartz_Cache_Source AND EVAPS2.PRM_SHUTTER_Option THEN
		IF EVAPS2.PRM_CTRL_DELAY_TIME = 0 THEN
			XTC3.I_Delay_Option		:=	1; (*shutter*)
		ELSE
			XTC3.I_Delay_Option		:=	3; (*both*)
			XTC3.I_Ctrl_Delay_Time	:=	EVAPS2.PRM_CTRL_DELAY_TIME;
		END_IF
		(*
		XTC3.I_Transfer_Sensor		:=	1;
		XTC3.I_Transfer_Tool			:=	EVAPS1.PRM_Transfer_Tooling;	(*Pas de 2eme sensor sous cache *)
		*)
	ELSE
		IF EVAPS2.PRM_CTRL_DELAY_TIME = 0 THEN
			XTC3.I_Delay_Option		:=	0; (*none*)
		ELSE
			XTC3.I_Delay_Option		:=	2; (*controle*)
			XTC3.I_Ctrl_Delay_Time	:=	EVAPS2.PRM_CTRL_DELAY_TIME;
		END_IF
		(*
		XTC3.I_Transfer_Sensor		:=	0;								(*Pas de 2eme sensor sous cache*)
		*)
	END_IF
END_IF

IF MAIN.STEP_EMPILEMENT.PRM_UTIL_SOURCE3 THEN
	XTC3.I_Soak_Power_2		:=	EVAPS3.PRM_SOAK2_POWER;
	XTC3.I_Deposition_Rate	:=	EVAPS3.PRM_Rate;
	XTC3.I_Thick_SP			:=	EVAPS3.PRM_Thick_SP;
	XTC3.I_New_Rate			:=	EVAPS3.PRM_New_Rate;
	XTC3.I_Rate_Ramp_Time	:=	EVAPS3.PRM_Rate_Ramp_Time;
	XTC3.I_Stab_Single		:=	EVAPS3.PRM_Stability_Single;
	XTC3.I_Stab_Total		:=	EVAPS3.PRM_Stability_Total;
	XTC3.I_Quality_Percent	:=	EVAPS3.PRM_Quality_Percent;
	XTC3.I_Quality_Counts	:=	EVAPS3.PRM_Quality_Counts;
	XTC3.I_PID_Gain			:=	EVAPS3.PRM_GAIN;
	XTC3.I_PID_Ti			:=	EVAPS3.PRM_INTEGRAL;
	XTC3.I_PID_Td			:=	EVAPS3.PRM_DERIVEE;
	XTC3.I_Max_Power		:=	EVAPS3.PRM_PMAX;
	IF EVAPS3.PRM_Quartz_Cache_Source AND EVAPS3.PRM_SHUTTER_Option THEN
		IF EVAPS3.PRM_CTRL_DELAY_TIME = 0 THEN
			XTC3.I_Delay_Option		:=	1; (*shutter*)
		ELSE
			XTC3.I_Delay_Option		:=	3; (*both*)
			XTC3.I_Ctrl_Delay_Time	:=	EVAPS3.PRM_CTRL_DELAY_TIME;
		END_IF
		(*
		XTC3.I_Transfer_Sensor		:=	1;
		XTC3.I_Transfer_Tool			:=	EVAPS1.PRM_Transfer_Tooling;	(*Pas de 2eme sensor sous cache *)
		*)
	ELSE
		IF EVAPS3.PRM_CTRL_DELAY_TIME = 0 THEN
			XTC3.I_Delay_Option		:=	0; (*none*)
		ELSE
			XTC3.I_Delay_Option		:=	2; (*controle*)
			XTC3.I_Ctrl_Delay_Time	:=	EVAPS3.PRM_CTRL_DELAY_TIME;
		END_IF
		(*
		XTC3.I_Transfer_Sensor		:=	0;								(*Pas de 2eme sensor sous cache*)
		*)
	END_IF
END_IF

TIMER_ECO_MODE(	IN:= ECO_MODE OR MACHINE.STATE_Off, 
				PT:= T#1M30S); 		(*Temps inhibition défaut lors de la sortie de veille*)

XTC3(
	MANUAL:= MACHINE.STATE_Manu,
	RESET:= MACHINE.STATE_Off,
	CO_START:= (MAIN.STEP_EMPILEMENT.PRM_UTIL_SOURCE1 AND EVAPS1.OUT_Start_Controleur AND NOT EVAPS1.PRM_PFixe)
					OR (MAIN.STEP_EMPILEMENT.PRM_UTIL_SOURCE2 AND EVAPS2.OUT_Start_Controleur AND NOT EVAPS2.PRM_PFixe)
					OR (MAIN.STEP_EMPILEMENT.PRM_UTIL_SOURCE3 AND EVAPS3.OUT_Start_Controleur AND NOT EVAPS3.PRM_PFixe),
	CO_STOP:= MAIN.STEP_EMPILEMENT.OUT_STOP_CONTROLEUR
					OR EXECPROC.STATE_INTERRUPTED
					OR INIT_MACHINE.RQ_STOP_CONTROLLER,
	CO_RAZ_THICK:= MAIN.STEP_EMPILEMENT.OUT_RAZ_THICK_CONTROLEUR,
	CO_RESET_Ctrl:= MAIN.STEP_EMPILEMENT.OUT_RESET_CONTROLEUR
					(*OR (MAIN.STEP_EMPILEMENT.PRM_UTIL_SOURCE1 AND EVAPS1.OUT_Start_Controleur AND EVAPS1.PRM_PFixe)
					OR (MAIN.STEP_EMPILEMENT.PRM_UTIL_SOURCE2 AND EVAPS2.OUT_Start_Controleur AND EVAPS2.PRM_PFixe)
					OR (MAIN.STEP_EMPILEMENT.PRM_UTIL_SOURCE3 AND EVAPS3.OUT_Start_Controleur AND EVAPS3.PRM_PFixe)*),
	CO_Enable:= MACHINE.STATE_On,
	CO_Load_Param:= MAIN.STEP_EMPILEMENT.RQ_LOAD_PARAM,
	I_Final_Thickness:= MAIN.STEP_EMPILEMENT.PRM_EPAISSEUR,
	I_Tool_Factor1:= MAIN.STEP_EMPILEMENT.PRM_TOOLING_QZ[0],
	I_Tool_Factor2:= MAIN.STEP_EMPILEMENT.PRM_TOOLING_QZ[1],
	I_Densite:= MAIN.STEP_EMPILEMENT.PRM_DENSITE_QZ[0],
	I_ZRatio:= MAIN.STEP_EMPILEMENT.PRM_ZRATIO_QZ[0],
	I_Time_Power:= MAIN.STEP_EMPILEMENT.PRM_TIMEPOWER, 
	I_Inhibe_Def:= TIMER_ECO_MODE.Q,);
	
(*Affectation des sorties*)
IF EXECPROC.RQ_FM_EXEC_STEP[17] OR (VISU_STOP_ECO_MANU AND MACHINE.STATE_Manu) THEN					(*début étape standby*)
	ECO_MODE := TRUE;
ELSIF EXECPROC.RQ_FM_EXEC_STEP[18] OR (NOT VISU_STOP_ECO_MANU AND MACHINE.STATE_Manu) THEN			(*fin étape standby*)
	ECO_MODE := FALSE;
ELSIF EXECPROC.OP_RUN.AR THEN
	ECO_MODE := MACHINE.RQ_Standby OR MACHINE.STATE_Standby;		(*dans ce cas c'est mode de marche qui prend la main*)
END_IF

OUT_MEG1 	:= NOT ECO_MODE AND PRG_POMPAGE.M11.STATE_Seuil[8];
OUT_MEJ1	:= SOURCE2.OUT_MEJ;
OUT_MEJ2	:= SOURCE3.OUT_MEJ;
IF SOURCE2.OUT_MEJ THEN
	OUT_QEJ1		:=	SOURCE2.OUT_QEJ;
ELSIF SOURCE3.OUT_MEJ THEN
	OUT_QEJ2		:=	SOURCE3.OUT_QEJ;
ELSE
	OUT_QEJ1		:=	0;
	OUT_QEJ2		:=	0;
END_IF
OUT_MPR230 	:= NOT ECO_MODE;

STATE_AR:= ((MACHINE.STATE_Auto OR MACHINE.STATE_Prod) AND EVAPS1.OP_Stop.OK AND EVAPS2.OP_Stop.OK AND EVAPS3.OP_Stop.OK) OR
			(MACHINE.STATE_MANU AND NOT SOURCE1.STATE_SRC
			AND NOT SOURCE1.STATE_HV AND NOT SOURCE2.STATE_EJ_ON AND NOT SOURCE3.STATE_EJ_ON  );

(*Défauts venant interrompre le procédé*)
STATE_Def_IProc := 	CC11.STATE_Nok OR
					CC12.STATE_Nok OR
					CC13.STATE_Nok OR
					EVAPS1.DEF_QZ_CTRL_RATE.DEF OR
					EVAPS1.DEF_Pmax.DEF OR
					EVAPS1.DEF_Pmin.DEF OR
					EVAPS1.DEF_TEMPS_MAX.DEF OR
					EVAPS1.DEF_REF.DEF OR
					EVAPS2.DEF_QZ_CTRL_RATE.DEF OR
					EVAPS2.DEF_Pmax.DEF OR
					EVAPS2.DEF_Pmin.DEF OR
					EVAPS2.DEF_TEMPS_MAX.DEF OR
					EVAPS2.DEF_REF.DEF OR
					EVAPS3.DEF_QZ_CTRL_RATE.DEF OR
					EVAPS3.DEF_Pmax.DEF OR
					EVAPS3.DEF_Pmin.DEF OR
					EVAPS3.DEF_TEMPS_MAX.DEF OR
					EVAPS3.DEF_REF.DEF OR
					SOURCE1.STATE_NOK OR
					SOURCE2.STATE_NOK OR
					SOURCE3.STATE_NOK OR
					XTC3.DEF_COM_STATUS.DEF OR
					XTC3.DEF_COM_PARAMETER.DEF OR
					XTC3.DEF_COM_COMMAND.DEF OR
					(QZ1.DEF_QZ.DEF AND NOT MODE_QUARTZ_PROD.STATE_Mode) OR //AND (NOT XTC3.I_Time_Power) OR //option time_power gérée dans l'XTC si tête rotary déclarée
					QZ1.DEF_Positionnement.DEF OR
					CRUCIBLE1.STATE_NOK;

END_FUNCTION_BLOCK

// ---- POUs/Composant/EVAP/BLOCK_XTAL6.TcPOU
FUNCTION_BLOCK BLOCK_XTAL6

(* Gestion d'une d'une tête multiquartz *)
(* Version 0 - SD- affaire 8152 *)
(* Version 1 - GV - 05/2015 - Correction Reset des G7 sur passage en manu - 8950*)

VAR_INPUT
	I_APPLY_PARAMETER:	BOOL;
	RESET:				BOOL;
	MANUAL:				BOOL;
	CTRL_PLC:			BOOL;

	IN_QF:				BOOL;		(*Quartz actif en panne*)
	IN_RATE:			REAL;		(*Vitesse de dépot mesurée sur le quartz acitf*)
	IN_FREQ:			REAL;		(*Frequence du quartz actif*)
	IN_THICKNESS:		REAL;		(*Epaisseur mesurée sur le quartz acitf*)
	IN_LIFE:			REAL;		(*Vie du quartz actif*)
	IN_ACTIVITY:		REAL;		(*Activité du quartz actif*)
	CO_SWITCH_CRYSTAL:	BOOL;		(*Pilotage Switch Crystal provenant de l'IC6*)

	CO_Positionnement:	BOOL;		(*Commande de positionnement de la tête MultiQuartz*)
	CO_Scan_Quartz:		BOOL;		(*Commande de scan des Quartz*)

	(*Consigne*)
	CONS_MATERIAL:	 	STRING;		(*Materiau*)
	CONS_POID:			REAL;		(*Poids du quartz pour la calcul du quartz*)
	CONS_ZRATIO:		REAL;		(*Valeur du Zratio*)
	CONS_DENSITE:		REAL;		(*Valeur de densité*)
	CONS_TOOLING:		REAL;		(*Facteur de correction de chaque quartz*)


	QZ11T		AT%I*:		BOOL;		(*Position sur Quartz n°1*)
	QZ12T		AT%I*:		BOOL;		(*Position sur Quartz n°2*)
	QZ13T		AT%I*:		BOOL;		(*Position sur Quartz n°3*)
	QZ14T		AT%I*:		BOOL;		(*Position sur Quartz n°4*)
	QZ15T		AT%I*:		BOOL;		(*Position sur Quartz n°5*)
	QZ16T		AT%I*:		BOOL;		(*Position sur Quartz n°6*)

(*Composant de la fonction*)
	QZ1_SWITCH:				BLOCK_ACTUATOR2;

(*défaut*)
	DEF_QZ:					PRCDEF;	(*Défaut quartz utilisé*)
	DEF_Positionnement:		PRCDEF;	(*Défaut de positionnement*)

(*Alarme*)
	ALM_SURV_ACTIVITY_QZ1:		PRCDEF;			(*Alarme surveillance activité du Quartz n°1*)
	ALM_SURV_ACTIVITY_QZ2:		PRCDEF;			(*Alarme surveillance activité du Quartz n°2*)
	ALM_SURV_ACTIVITY_QZ3:		PRCDEF;			(*Alarme surveillance activité du Quartz n°3*)
	ALM_SURV_ACTIVITY_QZ4:		PRCDEF;			(*Alarme surveillance activité du Quartz n°4*)
	ALM_SURV_ACTIVITY_QZ5:		PRCDEF;			(*Alarme surveillance activité du Quartz n°5*)
	ALM_SURV_ACTIVITY_QZ6:		PRCDEF;			(*Alarme surveillance activité du Quartz n°6*)

	ALM_SURV_LIFE_QZ1:			PRCDEF;			(*Alarme surveillance vie du Quartz n°1*)
	ALM_SURV_LIFE_QZ2:			PRCDEF;			(*Alarme surveillance vie du Quartz n°2*)
	ALM_SURV_LIFE_QZ3:			PRCDEF;			(*Alarme surveillance vie du Quartz n°3*)
	ALM_SURV_LIFE_QZ4:			PRCDEF;			(*Alarme surveillance vie du Quartz n°4*)
	ALM_SURV_LIFE_QZ5:			PRCDEF;			(*Alarme surveillance vie du Quartz n°5*)
	ALM_SURV_LIFE_QZ6:			PRCDEF;			(*Alarme surveillance vie du Quartz n°6*)

(*Opérations*)
	OP_Scan_Quartz:				BLOCK_OPERATION;	(* G7 de scan de l'état des quartz*)
	OP_Positionnement:			BLOCK_OPERATION;	(*G7 de positionnement du Quartz*)

(*Paramètres*)
	PRM_CONS_POSITION_QZ:		INT;		(*Consigne de position du Quartz*)

END_VAR
VAR_OUTPUT

	STATE_FREQUENCY:		ARRAY[0..6] OF REAL;	 (*Fréquence des quartz*)
	STATE_LIFE:				ARRAY[0..6] OF REAL; 	(*Vie des quartz*)
	STATE_ACTIVITY:			ARRAY[0..6] OF REAL;	(*Actvité des Quartz*)

	STATE_QF1:			BOOL;			(*Etat du Crystal 1*)
	STATE_QF2:			BOOL;			(*Etat du Crystal 2*)
	STATE_QF3:			BOOL;			(*Etat du Crystal 3*)
	STATE_QF4:			BOOL;			(*Etat du Crystal 4*)
	STATE_QF5:			BOOL;			(*Etat du Crystal 5*)
	STATE_QF6:			BOOL;			(*Etat du Crystal 6*)

	STATE_POSITION:		INT;				(*Position actuel du Quartz*)

	STATE_SCAN_QZ_AR:			BOOL;			(*Scan OK*)
	STATE_SCAN_QZ_EC:			BOOL;			(*Scan en cours*)
	STATE_POS_QZ_AR:			BOOL;			(*Positionnement OK*)
	STATE_POS_QZ_EC:			BOOL;			(*Positionnement en cours*)
	STATE_SELECT_QZ_OK:			BOOL;			(*Indique que la selection du Quartz est OK*)

	STATE_THICKNESS:			REAL;
	STATE_RATE:					REAL;
	STATE_MATERIAL:				STRING;
	STATE_NOK:					BOOL;

	STATE_ACTUAL_CRYS_FREQ:		REAL;
	STATE_ACTUAL_CRYS_LIFE:		REAL;
	STATE_ACTUAL_CRYS_ACTIVITY:	REAL;

	OUT_MATERIAL:				STRING;
	OUT_POIDS:					REAL;
	OUT_ZRATIO:					REAL;
	OUT_DENSITE:				REAL;
	OUT_TOOLING:				REAL;

	RQ_SWITCH_CRYSTAL:			BOOL;			(*Demande de Switch à une position donnée de la tête multiquartz*)
	OUT_CONS_POS_QUARTZ:		INT;				(*Consigne de position *)

	OUT_QZ1	AT %Q*:				BOOL;			(*Sortie Switch Crystal*)
END_VAR
VAR_INPUT PERSISTENT
	(*Entité*)
	IsComponent:	BOOL;			(*entité : composant*)
	IdXML:			STRING;			(*nom entité : identifiant pour recherche dans dico*)
	TagXML:			UINT;			(*nom entité : identifiant pour recherche dans dico*)
	IdParent:		STRING;			(*MNEMO de l'appelant*)
	MNEMO:			STRING;			(*MNEMO de l'entité*)

	PRM_Seuil_Life:			REAL;	(*Seuil d'alarme pour la vie du quartz*)
	PRM_Seuil_Activity:		REAL;	(*Seuil d'alarme pour l'activité du quartz*)

END_VAR
VAR
	VAR_Compteur:			INT;		(*Variable d'itération pour tête 6 Quartz*)
	MEM_POSITION_SCAN:		INT;		(*Variable mémoire position tête quartz*)
	MEM_POSITION:			INT;
	TIMER_Acq_Scan:			TON;	(*Timer d'acquisition du scan*)
	TIMER_Positionnement:	TON;	(*Timer de positionnement*)

	FM_Scan:				R_TRIG;
	FM_Etape_1_Position:	R_TRIG;
	VAR_Dmde_Scan:			BOOL;
	I:						INT;		(*Variable d'incrementation*)
END_VAR

PRL();

ACT_POSITIONNEMENT();
ACT_SCAN_QUARTZ();

POST();

ACTION ACT_POSITIONNEMENT:
(*Opération de Scan de l'état des Quartz*)
OP_Positionnement(
	CTRL_PLC:= CTRL_PLC,
	RESET:= RESET,
	ENABLE_INT:= OP_Scan_Quartz.Etape.0,
	MANUAL:= MANUAL,
	ON_AUTO_INT:=FALSE,
	RESTART_ENABLE_IF_OK:= TRUE,
	N_STEP_OP_OK:= 3,
	N_STEP_OP_NOK:=0 );

OP_Positionnement.PRL();

(*GRAFCET*)
(* initialisation du grafcet*)
IF 		OP_Positionnement.Etape = 0 THEN
				OP_Positionnement.Etape.0:=TRUE;

(*repositionnement sur étape 0*)
ELSIF MANUAL OR RESET
		THEN
				OP_Positionnement.Etape := 0;
				OP_Positionnement.Etape.0 := TRUE;

(*Etape 0-1*)
ELSIF	OP_Positionnement.Etape.0
		AND OP_Positionnement.MARCHE_OP
		AND OP_Scan_Quartz.Etape.0
		AND (PRM_CONS_POSITION_QZ>0)  THEN
				MEM_POSITION:= STATE_POSITION;
				OP_Positionnement.Etape.1:= TRUE;
				OP_Positionnement.Etape.0:= FALSE;

(*Etape 1-3*)
ELSIF	OP_Positionnement.Etape.1
		AND (STATE_POSITION = PRM_CONS_POSITION_QZ)  THEN
				OP_Positionnement.Etape.3:= TRUE;
				OP_Positionnement.Etape.1:= FALSE;

(*Rotation séquentielle*)
(*Etape 1-2*)
ELSIF	OP_Positionnement.Etape.1
		AND (STATE_POSITION <> MEM_POSITION) THEN
				MEM_POSITION:= STATE_POSITION;
				OP_Positionnement.Etape.2:= TRUE;
				OP_Positionnement.Etape.1:= FALSE;

(*Etape 2-3*)
ELSIF	OP_Positionnement.Etape.2
		AND (STATE_POSITION = PRM_CONS_POSITION_QZ)  THEN
				OP_Positionnement.Etape.3:= TRUE;
				OP_Positionnement.Etape.2:= FALSE;


(*Etape 2-1*)
ELSIF	OP_Positionnement.Etape.2
		AND (STATE_POSITION <> PRM_CONS_POSITION_QZ)
		AND TIMER_Positionnement.Q
		 THEN
				OP_Positionnement.Etape.1:= TRUE;
				OP_Positionnement.Etape.2:= FALSE;


ELSIF	OP_Positionnement.Etape.3
		AND (STATE_POSITION = PRM_CONS_POSITION_QZ)  THEN
				OP_Positionnement.Etape.0:= TRUE;
				OP_Positionnement.Etape.3:= FALSE;

END_IF

OP_Positionnement.POST();
END_ACTION

ACTION ACT_SCAN_QUARTZ:
(*Opération de Scan de l'état des Quartz*)
OP_Scan_Quartz(
	CTRL_PLC:= CTRL_PLC,
	RESET:= RESET,
	ENABLE_INT:=OP_Positionnement.Etape.0,
	MANUAL:= MANUAL,
	ON_AUTO_INT:=FALSE,
	RESTART_ENABLE_IF_OK:= TRUE,
	N_STEP_OP_OK:= 4,
	N_STEP_OP_NOK:=0 );

OP_Scan_Quartz.PRL();

(*GRAFCET*)
(* initialisation du grafcet*)
IF 		OP_Scan_Quartz.Etape = 0 THEN
				OP_Scan_Quartz.Etape.0:=TRUE;

(*repositionnement sur étape 0*)
ELSIF MANUAL OR RESET
		THEN
				OP_Scan_Quartz.Etape := 0;
				OP_Scan_Quartz.Etape.0 := TRUE;

(*Etape 0-1*)
ELSIF	OP_Scan_Quartz.Etape.0
		AND OP_Scan_Quartz.MARCHE_OP AND OP_Positionnement.Etape.0 THEN
				(*Mémorisation de la position du Quartz*)
				MEM_POSITION:= STATE_POSITION;
				VAR_Compteur:= 1;
				OP_Scan_Quartz.Etape.1:= TRUE;
				OP_Scan_Quartz.Etape.0:= FALSE;

(*Etape 1-2*)
ELSIF	OP_Scan_Quartz.Etape.1
		AND (STATE_POSITION<> MEM_POSITION) THEN
				MEM_POSITION:= STATE_POSITION;
				OP_Scan_Quartz.Etape.2:= TRUE;
				OP_Scan_Quartz.Etape.1:= FALSE;

(*Attente avant stablisation de la mesure*)
(*étape 2-3*)
ELSIF	OP_Scan_Quartz.Etape.2
		AND TIMER_Acq_Scan.Q THEN
				OP_Scan_Quartz.Etape.3:= TRUE;
				OP_Scan_Quartz.Etape.2:= FALSE;

(*étape 3-1*)
ELSIF	OP_Scan_Quartz.Etape.3
		AND VAR_Compteur<6 THEN
				VAR_Compteur:= VAR_Compteur + 1;
				OP_Scan_Quartz.Etape.1:= TRUE;
				OP_Scan_Quartz.Etape.3:= FALSE;

(*étape 3-4*)
ELSIF	OP_Scan_Quartz.Etape.3
		AND VAR_Compteur>=6 THEN
				VAR_Dmde_Scan:= FALSE;
				OP_Scan_Quartz.Etape.4:= TRUE;
				OP_Scan_Quartz.Etape.3:= FALSE;

ELSIF OP_Scan_Quartz.Etape.4 THEN
				OP_Scan_Quartz.Etape.0:= TRUE;
				OP_Scan_Quartz.Etape.4:= FALSE;


END_IF

OP_Scan_Quartz.POST();
END_ACTION

ACTION POST:
(*Position de la tête MultiQuartz*)
IF QZ11T THEN
	STATE_POSITION:=1;
ELSIF QZ12T THEN
	STATE_POSITION:=2;
ELSIF QZ13T THEN
	STATE_POSITION:=3;
ELSIF QZ14T THEN
	STATE_POSITION:=4;
ELSIF QZ15T THEN
	STATE_POSITION:=5;
ELSIF QZ16T THEN
	STATE_POSITION:=6;
END_IF

(*Gestion du changement de position du crystal*)
QZ1_SWITCH(
	RESET:= RESET,
	MANUAL:=MANUAL ,
	CO_On:=   CO_SWITCH_CRYSTAL ,
	EN_On_INT:= TRUE,
	EN_Off_INT:= TRUE,
	EN_On_EXT:= TRUE,			(*TOCHECK*)
	EN_Off_EXT:= TRUE,
	OUT_On=> OUT_QZ1,);

OUT_QZ1:=CO_SWITCH_CRYSTAL;
(*Demande de switch*)
RQ_SWITCH_CRYSTAL:= (OP_Positionnement.Etape.1 AND STATE_POSITION <> PRM_CONS_POSITION_QZ) OR OP_Scan_Quartz.Etape.1;

(*Acquisition des données du scan*)
IF OP_Scan_Quartz.Etape.3 OR OP_Positionnement.Etape.0 THEN
	CASE STATE_POSITION OF
		1:
			STATE_FREQUENCY[1]:= IN_FREQ;
			STATE_LIFE[1]:= IN_LIFE;
			STATE_ACTIVITY[1]:= IN_ACTIVITY;
			STATE_QF1:= IN_QF ;
		2:
			STATE_FREQUENCY[2]:= IN_FREQ;
			STATE_LIFE[2]:= IN_LIFE;
			STATE_ACTIVITY[2]:= IN_ACTIVITY;
			STATE_QF2:= IN_QF ;
		3:
			STATE_FREQUENCY[3]:= IN_FREQ;
			STATE_LIFE[3]:= IN_LIFE;
			STATE_ACTIVITY[3]:= IN_ACTIVITY;
			STATE_QF3:= IN_QF;
		4:
			STATE_FREQUENCY[4]:= IN_FREQ;
			STATE_LIFE[4]:= IN_LIFE;
			STATE_ACTIVITY[4]:= IN_ACTIVITY;
			STATE_QF4:= IN_QF;
		5:
			STATE_FREQUENCY[5]:= IN_FREQ;
			STATE_LIFE[5]:= IN_LIFE;
			STATE_ACTIVITY[5]:= IN_ACTIVITY;
			STATE_QF5:= IN_QF ;
		6:
			STATE_FREQUENCY[6]:= IN_FREQ;
			STATE_LIFE[6]:= IN_LIFE;
			STATE_ACTIVITY[6]:= IN_ACTIVITY;
			STATE_QF6:= IN_QF ;
	END_CASE
END_IF

(*Timer acquisition état des quartz*)
TIMER_Acq_Scan(
	IN := OP_Scan_Quartz.Etape.2,
	PT := T#10s
	 );


(*Timer acquisition état des quartz*)
TIMER_Positionnement(
	IN := OP_Positionnement.Etape.2,
	PT := T#10s
	 );

IF I_APPLY_PARAMETER THEN
	OUT_DENSITE 		:=		CONS_DENSITE;
	OUT_POIDS			:=		CONS_POID;
	OUT_ZRATIO		:=		CONS_ZRATIO;
	OUT_MATERIAL 		:= 		CONS_MATERIAL;
	OUT_TOOLING		:=		CONS_TOOLING;
END_IF

STATE_RATE:= 			IN_RATE;
STATE_THICKNESS:= 	IN_THICKNESS;
STATE_MATERIAL:=		OUT_MATERIAL;
STATE_NOK	:=			DEF_QZ.DEF;

(*Rotation séquentielle de la position*)
OUT_CONS_POS_QUARTZ:=0;


STATE_POS_QZ_AR:= NOT OP_Positionnement.Etape.1;
STATE_POS_QZ_EC:= OP_Positionnement.Etape.1;
STATE_SCAN_QZ_AR:= NOT OP_Scan_Quartz.Etape.1;
STATE_SCAN_QZ_EC:= OP_Scan_Quartz.Etape.1;

STATE_ACTUAL_CRYS_FREQ:= IN_FREQ;
STATE_ACTUAL_CRYS_LIFE:= IN_LIFE;
STATE_ACTUAL_CRYS_ACTIVITY:= IN_ACTIVITY;

(*Indique si la selection du quartz est ok*)
IF (STATE_POSITION = PRM_CONS_POSITION_QZ) AND STATE_POS_QZ_AR THEN
	STATE_SELECT_QZ_OK:=TRUE;
ELSE
	STATE_SELECT_QZ_OK:=FALSE;
END_IF


(*Alarme activité des quartz*)
ALM_SURV_ACTIVITY_QZ1(CONDITION := STATE_ACTIVITY[1] < PRM_Seuil_Activity, VAL1:= '1');
ALM_SURV_ACTIVITY_QZ2(CONDITION := STATE_ACTIVITY[2] < PRM_Seuil_Activity, VAL1:= '2');
ALM_SURV_ACTIVITY_QZ3(CONDITION := STATE_ACTIVITY[3] < PRM_Seuil_Activity, VAL1:= '3');
ALM_SURV_ACTIVITY_QZ4(CONDITION := STATE_ACTIVITY[4] < PRM_Seuil_Activity, VAL1:= '4');
ALM_SURV_ACTIVITY_QZ5(CONDITION := STATE_ACTIVITY[5] < PRM_Seuil_Activity, VAL1:= '5');
ALM_SURV_ACTIVITY_QZ6(CONDITION := STATE_ACTIVITY[6] < PRM_Seuil_Activity, VAL1:= '6');

(*Alarme vie des quartz*)
ALM_SURV_LIFE_QZ1(CONDITION:=STATE_LIFE[1] > PRM_Seuil_Life, VAL1:= '1');
ALM_SURV_LIFE_QZ2(CONDITION:=STATE_LIFE[2] > PRM_Seuil_Life, VAL1:= '2');
ALM_SURV_LIFE_QZ3(CONDITION:=STATE_LIFE[3] > PRM_Seuil_Life, VAL1:= '3');
ALM_SURV_LIFE_QZ4(CONDITION:=STATE_LIFE[4] > PRM_Seuil_Life, VAL1:= '4');
ALM_SURV_LIFE_QZ5(CONDITION:=STATE_LIFE[5] > PRM_Seuil_Life, VAL1:= '5');
ALM_SURV_LIFE_QZ6(CONDITION:=STATE_LIFE[6] > PRM_Seuil_Life, VAL1:= '6');



(*Défaut du Quartz utilisé, on vérifie que le positionnement n'est pas en cours et que c'est bien le Quartz utilisé qui est en défaut*)
DEF_QZ(
		CONDITION:=	IN_QF AND (STATE_POSITION = PRM_CONS_POSITION_QZ) AND STATE_POS_QZ_AR ,
		DELAY:=			T#10s);

(*Défaut de positionnement de la tête multiquartz*)
DEF_Positionnement(
		CONDITION:= OP_Positionnement.Etape.1 OR OP_Scan_Quartz.Etape.1,
		DELAY:=			T#30s);
END_ACTION

ACTION PRL:
TagXML:= 9;
IdXML:=	'16';

(*Défaut*)
DEF_QZ.IdXML := '14';
DEF_QZ.TagXML := 3;

DEF_Positionnement.IdXML := '14';
DEF_Positionnement.TagXML := 2;

(*Alarme*)
ALM_SURV_ACTIVITY_QZ1.IdXML:= '14';
ALM_SURV_ACTIVITY_QZ1.TagXML:= 15;
ALM_SURV_ACTIVITY_QZ1.Groupe := 1;

ALM_SURV_ACTIVITY_QZ2.IdXML:= '14';
ALM_SURV_ACTIVITY_QZ2.TagXML:= 15;
ALM_SURV_ACTIVITY_QZ2.Groupe := 1;

ALM_SURV_ACTIVITY_QZ3.IdXML:= '14';
ALM_SURV_ACTIVITY_QZ3.TagXML:= 15;
ALM_SURV_ACTIVITY_QZ3.Groupe := 1;

ALM_SURV_ACTIVITY_QZ4.IdXML:= '14';
ALM_SURV_ACTIVITY_QZ4.TagXML:= 15;
ALM_SURV_ACTIVITY_QZ4.Groupe := 1;

ALM_SURV_ACTIVITY_QZ5.IdXML:= '14';
ALM_SURV_ACTIVITY_QZ5.TagXML:= 15;
ALM_SURV_ACTIVITY_QZ5.Groupe := 1;

ALM_SURV_ACTIVITY_QZ6.IdXML:= '14';
ALM_SURV_ACTIVITY_QZ6.TagXML:= 15;
ALM_SURV_ACTIVITY_QZ6.Groupe := 1;

ALM_SURV_LIFE_QZ1.IdXML := '14';
ALM_SURV_LIFE_QZ1.TagXML := 16;
ALM_SURV_LIFE_QZ1.Groupe := 1;

ALM_SURV_LIFE_QZ2.IdXML := '14';
ALM_SURV_LIFE_QZ2.TagXML := 16;
ALM_SURV_LIFE_QZ2.Groupe := 1;

ALM_SURV_LIFE_QZ3.IdXML := '14';
ALM_SURV_LIFE_QZ3.TagXML := 16;
ALM_SURV_LIFE_QZ3.Groupe := 1;

ALM_SURV_LIFE_QZ4.IdXML := '14';
ALM_SURV_LIFE_QZ4.TagXML := 16;
ALM_SURV_LIFE_QZ4.Groupe := 1;

ALM_SURV_LIFE_QZ5.IdXML := '14';
ALM_SURV_LIFE_QZ5.TagXML := 16;
ALM_SURV_LIFE_QZ5.Groupe := 1;

ALM_SURV_LIFE_QZ6.IdXML := '14';
ALM_SURV_LIFE_QZ6.TagXML := 16;
ALM_SURV_LIFE_QZ6.Groupe := 1;


(*Switch Crystal QZ1*)
QZ1_SWITCH.CONF_Tim_Valid_Off		:=	T#0ms;
QZ1_SWITCH.CONF_Tim_Valid_On		:=	T#0ms;
QZ1_SWITCH.MNEMO					:=	'SQZ1';
QZ1_SWITCH.CONF_EN_On				:=	0;
QZ1_SWITCH.CONF_No_Safety_Auto		:=	FALSE;
QZ1_SWITCH.IdXML					:=	'4';
QZ1_SWITCH.TagXML					:=	1;
QZ1_SWITCH.IdParent					:=	MNEMO;
QZ1_SWITCH.DEF_Off_auto.IdXML		:=	'3';
QZ1_SWITCH.DEF_Off_auto.TagXML		:=	11;
QZ1_SWITCH.DEF_Off_Imposs.IdXML		:=	'3';
QZ1_SWITCH.DEF_Off_Imposs.TagXML	:=	9;
QZ1_SWITCH.DEF_On_Imposs.IdXML		:=	'3';
QZ1_SWITCH.DEF_On_Imposs.TagXML		:=	6;
END_ACTION

END_FUNCTION_BLOCK

// ---- POUs/Composant/BLOCK_ACTUATOR2.TcPOU
FUNCTION_BLOCK BLOCK_ACTUATOR2
(* Gestion d'un actionneur monostable sans retour *)

(****************historique des versions*****************************)

(* Version 1-0 - SP - VERSION INIITIALE 6844 DP650 N35*)
(* Version 2-0 - HG - Adaptation pour journal des évènements externe - 24/06/2011*)

(*************************************************************************)

VAR_INPUT
	I_PARAM_SYSTEM_OK:			BOOL;		(*paramétrage système ok*)
(*paramètre standard*)
	RESET:   					BOOL; 		(*Condition RAZ actionneur*)
	MANUAL:  					BOOL; 		(*Mode manuel*)
(*défaut du bloc*)
	DEF_On_Imposs:				PRCDEF;	(*04 - Défaut d'activation non autorisé en mode automatique*)
	DEF_Off_Imposs:				PRCDEF;	(*05 - Défaut de désactivation non autorisée en mode automatique*)
	DEF_Off_auto:				PRCDEF;	(*06 - Défaut de désactivation automatique*)

(*parametre de pilotage en entrée*)
	CO_On:   					BOOL; 			(*Ordre mode automatique activation*)
	EN_On_INT:   				BOOL:=TRUE;	(*Condition d'autorisation d'activation donnée par le bloc qui instancie le bloc actuator*)
	EN_Off_INT:  				BOOL:=TRUE; 	(*Condition d'autorisation de désactivation donnée par le bloc qui instacie le bloc actuator*)
	EN_On_EXT:					BOOL:=TRUE;	(*condition d'autorisation d'activation externe*)
	EN_Off_EXT:					BOOL:=TRUE;	(*condition d'autorisation de desactivation externe*)

	VAR_CPT:					BLOCK_CPT_APP;
END_VAR

VAR_INPUT PERSISTENT
(*parametre de configuration constructeur*)
(*les parametres suivants dépendent de la configuration de la machine*)
	CONF_No_Safety_Auto:		BOOL:=FALSE;	(*option de desactivation des conditions d'autorisation en mode automatique*)
	CONF_EN_On:					USINT:=0;		(*définit la réaction du système en cas de perte des conditions d'autorisation d'activation EN_On*)
												(* 0 = désactivation automatique  en cas de perte des conditions d'autorisation d'activation uniquement en manuel*)
												(* 1 = désactivation automatique en cas de perte des conditions d'autorisation d'activation en auto et en manuel*)
												(* 2 = Pas de déscativation automatique*)
	CONF_Tim_Valid_On:  		TIME; 			(*Temps validation actionneur on*)
	CONF_Tim_Valid_Off:   		TIME; 			(*Temps validation actionneur off *)

	(*Entité*)
	IsComponent:		BOOL;			(*entité : composant*)
	IdXML:				STRING;			(*nom entité : identifiant pour recherche dans dico*)
	TagXML:				UINT;			(*nom entité : identifiant pour recherche dans dico*)
	IdParent:			STRING;			(*MNEMO de l'appelant*)
	MNEMO:				STRING;			(*MNEMO de l'entité*)
END_VAR

VAR_OUTPUT
	OUT_On:				BOOL;	(*SORTIE TOR ACTIVATION*)
	STATE_On:	   		BOOL; 	(*Indicateur activation ok*)
	STATE_Off:  		BOOL; 	(*Indicateur désactivation ok*)
	STATE_Nok:			BOOL;	(*Indicateur défaut sur l'actionneur*)
	AUTOR_On_IHM:		BOOL; 	(*etat activation autorisée depuis la supervision*)
	AUTOR_Off_IHM:		BOOL; 	(*etat désactivation autorisée depuis la supervision*)
	AUTOR_On_PLC:		BOOL;	(*etat activation autorisée depuis l'automate*)
	AUTOR_Off_PLC:		BOOL;	(*etat désactivation autorisée depuis l'automate*)
END_VAR


VAR
	M_On:  				BOOL; 	(*Ordre mode manuel activation ou activation/desactivation si la vanne est monostable*)
	RCP_M_On:   		BOOL;
	VAR_On:				BOOL;	(*variable intermédiaire avant affectation de la sortie OUT_On *)

	TIMER_Valid_On:		TON;
	TIMER_Valid_Off:	TON;


END_VAR

VAR_EXTERNAL
	MANUAL_SAFETY_OFF:	BOOL;	(*desactive les sécurités en mode manuel*)
END_VAR

(* Réception des ordres en mode manuel*)
RCP_M_On 			:=	M_On;
(*Autorisation*)
AUTOR_On_IHM		:= 	MANUAL AND ((EN_On_INT AND EN_On_EXT)
						OR MANUAL_SAFETY_OFF) AND NOT RESET AND NOT VAR_On;
AUTOR_Off_IHM		:= 	MANUAL AND ((EN_Off_INT AND EN_Off_EXT)  OR
						MANUAL_SAFETY_OFF) AND NOT RESET AND  VAR_On;
AUTOR_On_PLC		:=	 NOT MANUAL AND ((EN_On_INT AND EN_On_EXT)
						OR CONF_No_Safety_Auto) AND NOT RESET;
AUTOR_Off_PLC		:= 	NOT MANUAL AND ((EN_Off_INT AND EN_Off_EXT)
						OR CONF_No_Safety_Auto) AND NOT RESET;

(*defaut activation impossible en mode automatique*)
DEF_On_Imposs.CONDITION:=	CO_On AND NOT AUTOR_On_PLC AND NOT RESET AND NOT MANUAL;
DEF_On_Imposs.DELAY := T#0ms;
DEF_On_Imposs();
(*Defaut désactivation impossible en mode automatique*)
DEF_Off_Imposs.CONDITION:=	NOT CO_On AND NOT AUTOR_Off_PLC
							AND NOT RESET AND NOT MANUAL;
DEF_Off_Imposs.DELAY := T#0ms;
DEF_Off_Imposs();
(*defaut desactivation automatique*)
DEF_Off_Auto.CONDITION :=        (NOT EN_On_INT OR NOT EN_On_EXT) AND  VAR_On AND ((CONF_En_ON=1) OR ((CONF_EN_On=0) AND MANUAL)) AND NOT RESET;
DEF_Off_auto.DELAY:=T#0ms;
DEF_Off_Auto();

(*gestion des sorties*)
IF 		(RCP_M_On AND AUTOR_On_IHM AND NOT VAR_ON) OR
		(CO_On AND AUTOR_On_PLC AND NOT VAR_ON) THEN
				VAR_On		:= 	TRUE;
ELSIF 	(RCP_M_On  AND VAR_ON  AND AUTOR_Off_IHM) OR
	    	(NOT CO_On AND VAR_ON AND AUTOR_Off_PLC) OR
		DEF_Off_Auto.DEF THEN
				VAR_On		:=	FALSE;
ELSIF 	RESET  THEN
				VAR_On		:= 	FALSE;
END_IF;
OUT_On			:=	VAR_On;

(*indicateur actionneur activé STATE_ON*)
TIMER_Valid_On.IN	:=	VAR_ON;
TIMER_Valid_On(PT:=CONF_Tim_Valid_On);
STATE_ON			:=	TIMER_Valid_On.Q;
(*indicateur actionneur activé STATE_OFF*)
TIMER_Valid_Off.IN	:=	NOT VAR_ON;
TIMER_Valid_Off(PT:=CONF_Tim_Valid_Off);
STATE_Off			:=	TIMER_Valid_Off.Q;

(*indicateur STATE_NOK*)
STATE_Nok			:=	DEF_On_Imposs.DEF OR DEF_OFF_auto.DEF ;


(*gestion compteur*)
VAR_CPT(I_On:= STATE_On);

(* Reset des ordres *)
IF M_On AND RCP_M_On THEN
	M_On 	:= FALSE;
END_IF;

END_FUNCTION_BLOCK

// ---- POUs/Fonction/FONCTIONS COMPTEUR/BLOCK_CPT_APP.TcPOU
FUNCTION_BLOCK BLOCK_CPT_APP
(* fonction permettant de compter un nombre d'apparition*)
(* il faut lier la variable Etat à la variable que l'on veut compter*)
(* la variable compteur donnera le nombre d'appartition de Etat depuis le début du lancement de la machine*)
(* la version initiale n'a pas été tracée*)
(*V2.0 - version initiale SP - 7326 - BA8*)
VAR_INPUT
	I_On:						BOOL;				(*donne si la fonction appelante est dans l'état marche (true) ou arret (false) *)
END_VAR
VAR
	FP_On:						R_TRIG;
END_VAR
VAR_INPUT PERSISTENT
	TagXML:						UINT;
	DISABLE:					BOOL;											(*indique que le compteur est desactivé*)
END_VAR
VAR PERSISTENT
	STATE_Cpt:	 				UDINT;				(*contient le nombre cumulé d'utilisation de la fonction*)
END_VAR

IF DISABLE THEN
	RETURN;
END_IF
FP_On(clk:=I_On);

IF FP_On.Q THEN
	STATE_Cpt	:=	STATE_Cpt + 1;
END_IF

END_FUNCTION_BLOCK

// ---- POUs/FONCTION DE BASE/BLOCK_OPERATION.TcPOU
FUNCTION_BLOCK BLOCK_OPERATION

(* Fonction de gestion d'une opération standard *)

(****************historique des versions******************************************************************************************************************)

(* Version 1-0 - SP - VERSION INIITIALE - 15/02/2010*)
(* Version 1-1 - SP - l'opération ne genère plud de défaut si une demande de marche depuis l'automate (ON_PLC) est générée et si l'opération est en cours ou
si l'opération est ok et que la marche de l'opération depuis l'état ok est autorisée*)
(* Version 2-0 - HG - Adaptation pour journal des évènements externe - 24/06/2011*)
(* Version 2.1 - SP - meilleur gestion du mem_on_ihm 17/11/2011 - SP - 7326 BA8*)

(**************************************************************************************************************************************************************)


VAR_INPUT
	(*condition en entrée*)
	ON_IHM:					BOOL;		(* ~ (OPC : 1 : available for OPC-clients) *)		(*ordre externe de	marche opération depuis l'IHM*)
	ON_PLC:					BOOL;						(*ordre interne de marche opération depuis l'automate*)
	ON_AUTO_INT:			BOOL;						(*condition interne à la fonction de déclenchement automatique de l'opération *)
	ON_AUTO_EXT:			BOOL;						(*condition externe à la fonction de déclenchement automatique de l'opération *)
	CTRL_PLC:				BOOL;						(*mode de contrôle de la fonction - 0 = contrôle depuis l'IHM - 1=contrôle depuis l'automate*)
	RESET:					BOOL;						(*condition de reset de la fonction*)
	MANUAL:					BOOL;						(*information de mode manuel*)
	ENABLE_EXT:				BOOL	:=TRUE;				(*condition externe à la fonction de marche de l'opération*)
	ENABLE_INT:				BOOL;						(*condition interne à la fonction de marche de l'opération*)
	RESTART_ENABLE_IF_OK:	BOOL;						(*le redémarrage de l'opération est autorisée si l'opération est à l'état OK*)
	N_STEP_OP_OK:			UINT (0..31);				(*n° d'étape correspondant à l'état OPERATION OK - 0 = inhibé*)
	N_STEP_OP_NOK:			UINT (0..31);				(*n° d'étape correspondant à l'état OPERATION NOK - 0 = inhibé*)

	(*information d'état*)
	AUTOR_IHM:					BOOL;		(* ~ (OPC : 1 : available for OPC-clients) *)		(*état marche opération depuis l'IHM autorisée*)

	AUTOR_PLC:					BOOL;		(* ~ (OPC : 1 : available for OPC-clients) *)		(*état marche opération depuis l'automate*)
	OK:							BOOL;		(* ~ (OPC : 1 : available for OPC-clients) *)		(*code d'état OK de l'opération*)
	EC:							BOOL;		(* ~ (OPC : 1 : available for OPC-clients) *)		(*code d'état EN COURS de l'opération*)
	AR:							BOOL;		(* ~ (OPC : 1 : available for OPC-clients) *)		(*code d'état de l'opération à l'ARRET*)
	NOK:						BOOL;		(* ~ (OPC : 1 : available for OPC-clients) *)		(*code d'état de l'opération Non OK*)
	MARCHE_OP:					BOOL;												(*bit de synthese de la demande de marche*)
	Etape:						UDINT;		(* ~ (OPC : 1 : available for OPC-clients) *)		(*étape du grafcet*)

	(*défaut*)
	DEF_AUTO_ON:				PRCDEF;											(*01 - défaut déclenchement automatique de l'opération*)
	DEF_ON_REJECTED:			PRCDEF;											(*02 - défaut marche opération refusé*)
END_VAR

VAR_OUTPUT
	STATUS:						UINT;		(* ~ (OPC : 1 : available for OPC-clients) *)		(*code d'état de l'opération*)
END_VAR

VAR
	I:					UINT;														(*variable d'itération*)
	FM_ON_AUTO_INT:	R_TRIG;														(*FM du bit ON_AUTO_INT*)
	FM_ON_AUTO_EXT:	R_TRIG;														(*FM du bit ON_AUTO_EXT*)
	FM_ON_PLC:		R_TRIG;														(*FM du bit de marche depuis l'automate*)
	MEM_ON_IHM:		BOOL;														(*bit mémoire de demande de marche depuis l'IHM*)
END_VAR

VAR_INPUT PERSISTENT
	(*Entité*)
	IsOperation:	BOOL;			(*entité : opération*)
	IdXML:			STRING;			(*nom entité : identifiant pour recherche dans dico*)
	TagXML:			UINT;			(*nom entité : identifiant pour recherche dans dico*)
	IdParent:		STRING;			(*MNEMO de l'appelant*)
	MNEMO:			STRING;			(*MNEMO de l'entité*)
END_VAR

DEF_AUTO_ON.IdXml			:=	'2';
DEF_AUTO_ON.TagXml			:=	2;

DEF_ON_REJECTED.IdXml		:=	'2';
DEF_ON_REJECTED.TagXml		:=	1;

ACTION POST:
(*renvoi du code d'état de l'opération*)
STATUS 	:= 		LREAL_TO_UINT(LN(UDINT_TO_REAL(etape)) / LN(2));

(*drapeau d'état de la fonction*)
OK		:=		(ETAPE=EXPT(2,N_STEP_OP_OK)) AND (N_STEP_OP_OK>0);
AR		:=		ETAPE.0;
EC 		:= 		NOT OK AND NOT AR;
NOK		:=		(ETAPE=EXPT(2,N_STEP_OP_NOK)) AND (N_STEP_OP_NOK>0) OR DEF_ON_REJECTED.APP;
END_ACTION

ACTION PRL:
MEM_ON_IHM := ON_IHM  ;								(*mémorisation de la demande IHM pour éviter les aléas*)

(*gestion front on_auto_int, on_auto_ext et on_int*)
FM_ON_AUTO_EXT(CLK:=ON_AUTO_EXT);
FM_ON_AUTO_INT(CLK:=ON_AUTO_INT);
FM_ON_PLC(CLK:=ON_PLC);


(*Opération autorisée en mode externe*)
AUTOR_IHM  	:=	NOT CTRL_PLC AND NOT MANUAL AND NOT RESET AND
					ENABLE_EXT AND (ETAPE.0 OR ((ETAPE=EXPT(2,N_STEP_OP_OK)) AND (N_STEP_OP_OK>0) AND RESTART_ENABLE_IF_OK))
					AND ENABLE_INT;

(*Opération autorisée en mode interne*)
AUTOR_PLC		:=	CTRL_PLC AND NOT MANUAL AND NOT RESET AND
					((ENABLE_EXT AND (ETAPE.0 OR ((ETAPE=EXPT(2,N_STEP_OP_OK)) AND (N_STEP_OP_OK>0) AND RESTART_ENABLE_IF_OK))
					AND ENABLE_INT)
					OR NOT (ETAPE.0 OR ((ETAPE=EXPT(2,N_STEP_OP_OK)) AND (N_STEP_OP_OK>0) AND RESTART_ENABLE_IF_OK)) )  ;

(*Affectation de la condition de marche et reset des ordres de marches interne et externe*)
MARCHE_OP	:=	(MEM_ON_IHM AND NOT CTRL_PLC  AND AUTOR_IHM) OR
					(FM_ON_PLC.Q AND CTRL_PLC AND AUTOR_PLC) OR
					(FM_ON_AUTO_INT.Q OR FM_ON_AUTO_EXT.Q) AND NOT RESET AND NOT MANUAL AND
										(ETAPE.0 OR ((ETAPE=EXPT(2,N_STEP_OP_OK)) AND (N_STEP_OP_OK>0) AND RESTART_ENABLE_IF_OK)) ;

(*Gestion du défaut de demande de marche opération refusée*)
DEF_ON_REJECTED.CONDITION 		:=	(MEM_ON_IHM AND NOT AUTOR_IHM) OR (FM_ON_PLC.Q AND NOT AUTOR_PLC);
DEF_ON_REJECTED.DELAY			:=	T#0s;
DEF_ON_REJECTED();
(*Gestion du défaut de déclenchement automatique de la fonction*)
DEF_AUTO_ON.CONDITION 			:=	(FM_ON_AUTO_INT.Q  OR FM_ON_AUTO_EXT.Q) AND NOT RESET AND NOT MANUAL AND
										(ETAPE.0 OR ((ETAPE=EXPT(2,N_STEP_OP_OK)) AND (N_STEP_OP_OK>0) AND RESTART_ENABLE_IF_OK)) ;
DEF_AUTO_ON.DELAY				:=	T#0s;
DEF_AUTO_ON();

(*RAZ des demande de marche PLC et IHM*)
IF ON_IHM AND MEM_ON_IHM THEN
	ON_IHM :=FALSE;
END_IF;
ON_PLC			:=	FALSE;
END_ACTION

END_FUNCTION_BLOCK

// ---- POUs/Fonction/ETHER COM/BLOCK_XTC3.TcPOU
FUNCTION_BLOCK BLOCK_XTC3
(*Fonction de communication Ethernet TCP/IP pour contrôleur de dépôt XTC3*)

(****************historique des versions*****************************)

(* Version 1-0 - SD - VERSION INITIALE - 8157 - 11/2013*)
(* Version 2-0 - SD - Ajout parametres rampe de prefusion - 8650 - 07/2014*)
(* Version 3-0 - GV/SP - Fiabilisation de la connexion/communication avec l'XTC*)
(* Version 4-0 - GV - Ajout CO_Switch_Crystal pour gestion tête multi-quartz - 8950 - 04/2015
				- Ajout attente serveur déconnecté dans G7 de gestion
				- Modification lancement des actions du G7 de gestion
				- Les commandes Start, Stop et Raz thickness sont maintenant envoyées par ethernet*)
(* Version 5-0 - GV - Optimisation temps processus + Modification condition défaut VAR_StatusReader  - 9070 - 09/2015*)
(* Version 5-1 - GV - Modification condition défaut VAR_ParameterWriter + VAR_CommandWriter - 10315 - 09\2017*)
(* Version 5-2 - GV - Ajout de la commande film to run = 1 - 08/2020*)
(* Version 5-3 - GV - Modification gestion STATE_READY + Ajout inhibition des défauts *)

(*Amélioration à prévoir*)
(*Voir pour tout envoyer d'un coup*)

(*************************************************************************)
VAR_INPUT
	MANUAL:					BOOL;
	RESET:						BOOL;						(* Condition de réinitialisation de la fonction *)
	CONF_sRemoteHost: 			STRING(15) := '192.168.0.20';	(* Adresse IP de l'XTC*)
	CONF_nRemotePort: 			UDINT := 2101;				(*N° de port de communication de l'XTC*)

(*Commande externe*)
	CO_START:					BOOL;	(*Demande de marche du contrôleur de dépôt*)
	CO_STOP:					BOOL;	(*Demande d'arrêt du contrôleur*)
	CO_RAZ_THICK:				BOOL;	(*Demande de RAZ épaisseur*)
	CO_RESET_Ctrl:				BOOL;	(*Demande de RESET du controleur*)
	CO_VALID_CREUSET:			BOOL;
	CO_Switch_Crystal:			BOOL;	(*Demande changement de quartz dans le cas d'une tête multi-quartz*)


	CO_Enable:					BOOL;	(* Demande d'activation de la communication, récupération automatique des valeurs de l'XTC*)
	CO_Load_Param:				BOOL;	(*Demande de chargement des parametres couche etc*)

	IN_CD31T	AT%I*:			BOOL;	(*Entrée XTC3 à l'état STOP*)
	IN_CD32T	AT%I*:			BOOL;	(*Entrée Fin de couche*)
	IN_CD33T	AT%I*:			BOOL;	(*Entrée Crystal Fail*)
	IN_CD34T	AT%I*:			BOOL;	(*Entrée Alarm*)

	IN_CD35T	AT%I*:			BOOL;	(*Entrée ouverture cache source*)
	IN_CD36T 	AT%I*:			BOOL;	(*Entrée ouverture cache Quartz*)

	IN_CD31Q	AT%I*:			INT;		(*Entrée analogique consigne puissance source*)

(*Action sur le controleur*)

(****Parametres chargés dans le contrôleur XTC3 avec la commande UF*)
	I_Rise_Time_1:			INT:=0;
	I_Soak_Power_1:			REAL:=0;
	I_Soak_Time_1:			INT:=0;
	I_Rise_Time_2:			INT:=0;
	I_Soak_Power_2:			REAL:=0;
	I_Soak_Time_2:			INT:=0;
	I_Idle_Ramp:				INT:=0;
	I_Idle_Power:				REAL:=0;
	I_Deposition_Rate:		REAL:=0;
	I_Final_Thickness:			REAL:=0;
	I_Thick_SP:				REAL:=0;		(*Epaisseur à partir duquel on applique la nouvelle consigne de vitesse*)
	I_New_Rate:				REAL:=0;		(*Nouvelle consigne de vitesse*)
	I_Rate_Ramp_Time:		UINT:=0;		(*Temps de montée pour la nouvelle vitesse*)
	I_Rate_Watcher_Accuracy:	INT:=1;
	I_RW_Hold_Time:			INT:=0;
	I_Sensor:				BYTE:=16#01;
	I_Tool_Factor1:			REAL:=100;	(*Facteur de correction crystal actif*)
	I_Tool_Factor2:			REAL:=100;	(*Facteur de correction crystal backup*)
	I_Stab_Single:			UINT:=0;
	I_Stab_Total:				UINT:=0;
	I_Quality_Percent:			USINT:=0;
	I_Quality_Counts:			USINT:=0;
	I_Source:				BYTE:=1;	(*Source à utiliser*)
	I_Crucible_Nb:			BYTE:=0;	(*Numéro de creuset à utiliser*)
	I_PID_Gain:				REAL:=1.0;	(*Gain PID*)
	I_PID_Ti:					REAL:=0.1;
	I_PID_Td:				REAL:=0.1;
	I_Max_Power:				REAL:=100.0;		(*Puissance max de la source*)
	I_Densite:				REAL:=1.0;		(*Densité du matériau utilisé en g/cc*)
	I_ZRatio:					REAL:=1.0;		(*Z-Ratio du matériau utilisé*)
	I_Time_Power:			BOOL:=FALSE;	(*Option TimePower = 1*)
	I_Delay_Option:			BYTE:=0;		(*Gestion de l'étalonnage de la vitesse d'évaporation, 0 =None, 1 = Shutter delay, 2 = Control, 3 = Both*)
	I_Transfer_Tool:			REAL:=100;
	I_Ctrl_Delay_Time:		INT:=0;
	I_Transfer_Sensor:		INT:=0;
	I_IAD_Deposit:			BOOL:=0;

(*opération*)
	OP_Gest:					BLOCK_G7; 	(*Opération de gestion Status, chargement parametres, Envoi de commandes*)

(*défaut*)
	DEF_COM_STATUS:			PRCDEF;	(*Défaut de communication port de lecture état de l'XTC*)
	DEF_COM_PARAMETER:		PRCDEF; 	(*Défaut de communication port écriture des paramètres de couche*)
	DEF_COM_COMMAND:		PRCDEF;	(*Défaut de communication port d'envoie de commande à l'XTC*)
	I_Inhibe_Def:			BOOL:=0;
END_VAR
VAR_OUTPUT
	(*Variable d'état de connextion*)
	hSocket:							T_HSOCKET; 	(*ID de connexion - *)

	(*Informations obtenues avec la commande S0*)
	STATE_Sensor_Fail:				BOOL;			(*Etat du Quartz , 0 = Good, 1 = Failed Crystal*)
	STATE_Phase:					STRING;			(*Phase du contrôleur, READY,DEPOSIT, etc*)
	STATE_NPhase:					BYTE;			(*Code de phase du controlleur*)
	STATE_Active_Sensor:			USINT;			(*Numéro du Capteur utilisé*)
	STATE_Active_Crystal:			USINT;			(*Numéro du Quartz utilisé pour un MultiQuartz*)
	STATE_Rate:						REAL;			(*Vitesse d'évaporation, A°/s*)
	STATE_Thickness:				REAL;			(*Epaisseur de dépôt, kA°*)
	STATE_Power:					REAL;			(*Puissance demandée en %*)
	STATE_Rate_Deviation:			REAL;			(*Rate deviation , A°/s*)
	STATE_Frequency:				REAL;			(*Fréquence du Quartz, Hz*)
	STATE_XTC_INPUT:				ARRAY[0..15] OF BOOL;	(*etat des entrrée de l'XTC*)
	STATE_Timer_Tick:				BYTE;			(*Dernière valeur connue du timer tick renvoyer dans les trames par l'XTC*)
	(*Information obtenues avec la commande S9*)
	STATE_Crystal_Life:				USINT;			(*Durée de vie du Crystal*)

	STATE_Prog_Layer_OK:			BOOL;			(*Indique que la programmation de la couche est OK*)
	STATE_NOK:						BOOL;			(*Driver en défaut*)
	STATE_READY:					BOOL;			(*Driver en fonctionnement*)
	STATE_ACTION_OK:				BOOL;			(*Indique que la demande d'action à été effectuée*)
	STATE_STOP:					BOOL;			(*Indique que le controleur est à l'état STOP*)

	STATE_START_OK:				BOOL;			(*TRUE lorsque la commande de start a été envoyée*)
	STATE_STOP_OK:				BOOL;			(*TRUE lorsque la commande de stop a été envoyée*)
	STATE_RESET_OK:				BOOL;			(*TRUE lorsque la commande de reset a été envoyée*)
	STATE_RAZ_THICK_OK:			BOOL;			(*TRUE lorsque la commande de raz thicknesse a été envoyée*)
	STATE_SWITCH_XTAL_OK:		BOOL;	 		(*TRUE lorsque la commande de switch est à OK*)

	(*Information en sortie de l'XTC3*)
	OUT_STOP_STATE:				BOOL;
	OUT_END_OF_PROCESS:			BOOL;
	OUT_CRYSTAL_FAIL:				BOOL;
	OUT_ALARMS:					BOOL;
	OUT_CACHE_SRCE:				BOOL;
	OUT_CACHE_QUARTZ:			BOOL;
	OUT_POWER_SP:				INT;

END_VAR
VAR

	VAR_StatusReader:					STRUCT_ClientConnect;	(*structure de variable associée à la lecture cyclique des états de l'XTC*)
	VAR_ParameterWriter:					STRUCT_ClientConnect;	(*structure de variable associée à la programmation des paramètres de l'XTC*)
	VAR_CommandWriter:					STRUCT_ClientConnect;	(*structure de variable associée à l'envoie de commande à l'XTC*)

(* Variables demande en mode manuel*)
	M_Start:						BOOL;	(*Ordre start en mode manuel*)
	M_Stop:						BOOL;	(*Ordre stop en mode manuel*)
	M_Reset:					BOOL;	(*Ordre reset en mode manuel*)
	M_RAZ_Thick:				BOOL;	(*Ordre raz epaisseur en mode manuel*)
	M_Load_param:				BOOL;	(*Ordre programmation de la couche en mode manuel*)
	M_Switch_Crystal:				BOOL;	(*Ordre de changement de quartz en mode manuel*)

	RCP_M_Start:					BOOL;	(*Reception ordre start en mode manuel*)
	RCP_M_Stop:				BOOL;	(*Reception ordre stop en mode manuel*)
	RCP_M_Reset:				BOOL;	(*Receptionordre reset en mode manuel*)
	RCP_M_RAZ_Thick:			BOOL;	(*Reception ordre raz epaisseur en mode manuel*)
	RCP_M_Load_param:			BOOL;	(*Reception ordre programmation de la couche en mode manuel*)
	RCP_M_Switch_Crystal:		BOOL;	(*Reception ordre de switch du crystal en mode manuel*)

	VAR_START:				BOOL;
	VAR_RAZ_THICK:				BOOL;
	VAR_STOP:					BOOL;
	VAR_LOAD_PARAM:			BOOL;
	VAR_RESET:				BOOL;
	VAR_SWITCH_CRYSTAL:		BOOL;

	FM_CO_Load_Param:			R_TRIG;	(*Gestion du front montant de la demande de paramétrage en automatique*)
	FM_CO_RESET_Ctrl:			R_TRIG; (*Gestion de front montant de la demande de reset en automatique*)
	FM_CO_Start:					R_TRIG;	(*Gestion de front montant de la demande de start en automatique*)
	FM_CO_Stop:					R_TRIG;	(*Gestion de front montant de la demande de stop en automatique*)
	FM_CO_Raz_Thick:			R_TRIG; (*Gestion de front montant de la demande de remise à zéro de l'épaisseur en automatique*)
	FM_CO_Switch_Crystal:		R_TRIG;	(*Gestion de front montant de la demande de changement quartz en automatique*)

	FD_Manual:					F_TRIG;	(*Gestion du front descendant du mode manuel*)

	TEMP_REAL:					REAL;
	TEMP_DWORD:				DWORD;

	VAR_Frequence:				ARRAY[0..7] OF BYTE;	(* 8 octets pour la fréquence de chaque Quartz*)

	VAR_Freq_Multiplieur:			REAL:=0.0034924596;	(*Facteur de conversion Fréquence(Hz)*)

	Def_connect_com_status:		BOOL;				(*Flag en cas de défaut de connection com_status*)
	Def_connect_com_parameters:	BOOL;				(*Flag en cas de défaut de connection com_parameters*)
	Def_connect_com_command:	BOOL;				(*Flag en cas de défaut de connection com_command*)
	Condition_def_com_status:		BOOL;				(*Condition d'apparition défaut com_satus*)
	Condition_def_com_parameters: BOOL;				(*Condition d'apparition défaut com_parameters*)
	Condition_def_com_command:	BOOL;				(*Condition d'apparition défaut com_command*)

	(*Visualisation TC3*)
	VISU_Show_Details:			BOOL;
	
	(*Timer validation STATE_Ready*)
	TIMER_STATE_READY:			TON;
END_VAR
VAR_INPUT PERSISTENT
	(*Entité*)
	IsComponent:		BOOL;			(*entité : composant*)
	IdXML:			STRING;			(*nom entité : identifiant pour recherche dans dico*)
	TagXML:			UINT;			(*nom entité : identifiant pour recherche dans dico*)
	IdParent:			STRING;			(*MNEMO de l'appelant*)
	MNEMO:			STRING;			(*MNEMO de l'entité*)
END_VAR

PRL();

(*Appel des processus de communication*)
VAR_StatusReader.ConnectTime := T#50ms;
VAR_StatusReader.ExchangeCycleTime := T#10ms;
COM_STATUS();

VAR_ParameterWriter.ConnectTime := T#1s;
VAR_ParameterWriter.ExchangeCycleTime := T#10ms;
COM_PARAM();

VAR_CommandWriter.ConnectTime := T#50ms;
VAR_CommandWriter.ExchangeCycleTime := T#10ms;
COM_COMMAND();

(*appel des opérations*)
ACT_GESTION();

(*action en sortie*)
POST();

ACTION ACT_GESTION:
OP_Gest(
	N_STEP_OP_OK:= 0,
	N_STEP_OP_NOK:=0 );


(*GRAFCET*)
(* initialisation du grafcet*)
IF 		OP_Gest.Etape = 0 THEN
				OP_Gest.Etape.0:=TRUE;
(*repositionnement sur étape 0*)
ELSIF RESET THEN
				OP_Gest.Etape := 0;
				OP_Gest.Etape.0 := TRUE;
(*étape 0-1*)
ELSIF OP_Gest.Etape.0
			AND VAR_ParameterWriter.eStep = CLIENT_STATE_IDLE
			AND VAR_CommandWriter.eStep = CLIENT_STATE_IDLE
			AND NOT VAR_ParameterWriter.bConnected
			AND NOT VAR_CommandWriter.bConnected
			THEN
				OP_Gest.Etape.1:= TRUE;
				OP_Gest.Etape.0:= FALSE;
(*étape 1-2*)
ELSIF OP_Gest.Etape.1
			AND VAR_LOAD_PARAM
			THEN
				OP_Gest.Etape.2 := TRUE;
				OP_Gest.Etape.1 := FALSE;
(*étape 2-3*)
ELSIF OP_Gest.Etape.2
			AND VAR_StatusReader.eStep = CLIENT_STATE_IDLE
			AND NOT VAR_StatusReader.bConnected
			THEN
				OP_Gest.Etape.3 := TRUE;
				OP_Gest.Etape.2 := FALSE;
(*étape 3-4*)
ELSIF OP_Gest.Etape.3
			AND (STATE_Prog_Layer_OK OR VAR_ParameterWriter.bError)
			THEN
				OP_Gest.Etape.4 := TRUE;
				OP_Gest.Etape.3 := FALSE;
(*étape 4-0*)
ELSIF OP_Gest.Etape.4 THEN
				OP_Gest.Etape.0 := TRUE;
				OP_Gest.Etape.4 := FALSE;
(*étape 1-5*)
ELSIF OP_Gest.Etape.1
			AND (VAR_START OR VAR_STOP OR VAR_RAZ_THICK OR VAR_RESET OR VAR_SWITCH_CRYSTAL)
			THEN
				OP_Gest.Etape.5 := TRUE;
				OP_Gest.Etape.1 := FALSE;
(*étape 5-6*)
ELSIF OP_Gest.Etape.5
			AND VAR_StatusReader.eStep = CLIENT_STATE_IDLE
			AND NOT VAR_StatusReader.bConnected
			THEN
				OP_Gest.Etape.6 := TRUE;
				OP_Gest.Etape.5 := FALSE;
(*étape 6-7*)
ELSIF OP_Gest.Etape.6
			AND (STATE_ACTION_OK OR VAR_CommandWriter.bError)
			THEN
				OP_Gest.Etape.7 := TRUE;
				OP_GEst.Etape.6 := FALSE;
(*étape 7-0*)
ELSIF OP_Gest.Etape.7 THEN
				OP_Gest.Etape.0 := TRUE;
				OP_Gest.Etape.7 := FALSE;
END_IF
END_ACTION

ACTION COM_COMMAND:
CASE VAR_CommandWriter.eStep OF
	CLIENT_STATE_IDLE:		(*Etape 0 - sequence d'échange à l'arrêt*)
		(*si demande de marche ou exclusif serveur connecté*)
		IF VAR_CommandWriter.bEnable XOR VAR_CommandWriter.bConnected THEN
			VAR_CommandWriter.bBusy := TRUE;
			VAR_CommandWriter.bError := FALSE;
			VAR_CommandWriter.nErrid := 0;
			(*si demande d'exécution des échanges et pas le serveur connecté - on demande la connexion*)
			IF VAR_CommandWriter.bEnable THEN
				VAR_CommandWriter.fbConnectTON( IN := FALSE );
				VAR_CommandWriter.eStep := CLIENT_STATE_CONNECT_START;
			(*sinon cad pas demande d'execution et que le serveur est connecté - on demande la fermeture du port*)
			ELSE
				VAR_CommandWriter.eStep := CLIENT_STATE_CLOSE_START;
			END_IF
		(*si connection demandé et serveur connecté - on passe directement au échange*)
		ELSIF VAR_CommandWriter.bConnected THEN
			VAR_CommandWriter.fbDataExchaTON( IN := FALSE );
			VAR_CommandWriter.eStep := CLIENT_STATE_DATAEXCHA_START;
		ELSE
			VAR_CommandWriter.bBusy := FALSE;
		END_IF

	CLIENT_STATE_CONNECT_START: (*Etape 1 - connexion au port*)
		(*temporisation de reconnexion*)
		VAR_CommandWriter.fbConnectTON( IN := TRUE, PT := VAR_CommandWriter.connectTime);
		(*si tempo de reconnexion ok*)
		IF VAR_CommandWriter.fbConnectTON.Q THEN
			VAR_CommandWriter.fbConnectTON( IN := FALSE );
			VAR_CommandWriter.fbConnect(  bExecute := FALSE  );
			VAR_CommandWriter.fbConnect(
						sRemoteHost		:= CONF_sRemoteHost,
						nRemotePort		:= CONF_nRemotePort,
						 sSrvNetId		:= '',
						bExecute		:= TRUE );
			VAR_CommandWriter.eStep := CLIENT_STATE_CONNECT_WAIT;
			VAR_CommandWriter.Compteur_connection := VAR_CommandWriter.Compteur_connection + 1;
		END_IF

	CLIENT_STATE_CONNECT_WAIT:	(*Etape 2 - attente connexion ok*)
		VAR_CommandWriter.fbConnect( bExecute := FALSE );
		IF NOT VAR_CommandWriter.fbConnect.bBusy THEN
			IF NOT VAR_CommandWriter.fbConnect.bError THEN
				VAR_CommandWriter.bConnected 	:= TRUE;
				VAR_CommandWriter.hSocket 	:= VAR_CommandWriter.fbConnect.hSocket;
				VAR_CommandWriter.eStep 	:= CLIENT_STATE_IDLE;
				Def_connect_com_command := FALSE;
				(*reinitalisation du n° de requete en fonction de la premier commande demandée dans l'ordre de transmission*)
				IF VAR_START THEN
					VAR_CommandWriter.nRequest := 0;
				ELSIF VAR_STOP THEN
					VAR_CommandWriter.nRequest := 1;
				ELSIF VAR_RESET THEN
					VAR_CommandWriter.nRequest := 2;
				ELSIF VAR_RAZ_THICK  THEN
					VAR_CommandWriter.nRequest := 3;
				ELSIF VAR_SWITCH_CRYSTAL THEN
					VAR_CommandWriter.nRequest := 4;
				(*si aucune commande active alors que le gracet a été lancé*)
				(*on repositionne en idle et on valide l'état state_action_ok pour ne pas bloquer le grafcet de gestion des échanges *)
				ELSE
					STATE_ACTION_OK := TRUE;
					VAR_CommandWriter.eStep := CLIENT_STATE_IDLE;
				END_IF
			ELSE
				VAR_CommandWriter.nErrId := VAR_CommandWriter.fbConnect.nErrId;
				VAR_CommandWriter.nStepInError  := 2;
				VAR_CommandWriter.ErrDescription := CONCAT('FbConnect Error : ', UDINT_TO_STRING(VAR_CommandWriter.fbConnect.nErrId));
				VAR_CommandWriter.eStep := CLIENT_STATE_ERROR;
				Def_connect_com_command := TRUE;
			END_IF
		END_IF

	CLIENT_STATE_DATAEXCHA_START:	(*Etape 3 - lancement des échanges*)
		VAR_CommandWriter.fbDataExchaTON( IN := TRUE, PT := VAR_CommandWriter.ExchangeCycleTime );
		IF VAR_CommandWriter.fbDataExchaTON.Q THEN
			VAR_CommandWriter.fbDataExchaTON( IN := FALSE );
			VAR_CommandWriter.fbClientDataExcha( bExecute := FALSE );

			CASE VAR_CommandWriter.nRequest  OF
			0:
				(*Start - R0*)
				VAR_CommandWriter.fbClientDataExcha.txBuffer[0]:=16#02;
				VAR_CommandWriter.fbClientDataExcha.txBuffer[1]:=16#00;
				VAR_CommandWriter.fbClientDataExcha.txBuffer[2]:= F_ToASC('R');
				VAR_CommandWriter.fbClientDataExcha.txBuffer[3]:= 16#00;
				VAR_CommandWriter.fbClientDataExcha.txBuffer[4]:= VAR_CommandWriter.fbClientDataExcha.txBuffer[2] +
															VAR_CommandWriter.fbClientDataExcha.txBuffer[3];
				VAR_CommandWriter.fbClientDataExcha.nbTransmittedChar := 5;
				VAR_CommandWriter.fbClientDataExcha.nbExpectedChar := 6;
			1:
				(*Stop - R1*)
				VAR_CommandWriter.fbClientDataExcha.txBuffer[0]:=16#02;
				VAR_CommandWriter.fbClientDataExcha.txBuffer[1]:=16#00;
				VAR_CommandWriter.fbClientDataExcha.txBuffer[2]:= F_ToASC('R');
				VAR_CommandWriter.fbClientDataExcha.txBuffer[3]:= 16#01;
				VAR_CommandWriter.fbClientDataExcha.txBuffer[4]:= VAR_CommandWriter.fbClientDataExcha.txBuffer[2] +
															VAR_CommandWriter.fbClientDataExcha.txBuffer[3];
				VAR_CommandWriter.fbClientDataExcha.nbTransmittedChar := 5;
				VAR_CommandWriter.fbClientDataExcha.nbExpectedChar := 6;
			2:
				(*Reset - R2*)
				VAR_CommandWriter.fbClientDataExcha.txBuffer[0]:=16#02;
				VAR_CommandWriter.fbClientDataExcha.txBuffer[1]:=16#00;
				VAR_CommandWriter.fbClientDataExcha.txBuffer[2]:= F_ToASC('R');
				VAR_CommandWriter.fbClientDataExcha.txBuffer[3]:= 16#02;
				VAR_CommandWriter.fbClientDataExcha.txBuffer[4]:= VAR_CommandWriter.fbClientDataExcha.txBuffer[2] +
															VAR_CommandWriter.fbClientDataExcha.txBuffer[3];
				VAR_CommandWriter.fbClientDataExcha.nbTransmittedChar := 5;
				VAR_CommandWriter.fbClientDataExcha.nbExpectedChar := 6;
			3:
				(*Raz Thick - 12*)
				VAR_CommandWriter.fbClientDataExcha.txBuffer[0]:=16#02;
				VAR_CommandWriter.fbClientDataExcha.txBuffer[1]:=16#00;
				VAR_CommandWriter.fbClientDataExcha.txBuffer[2]:= F_ToASC('R');
				VAR_CommandWriter.fbClientDataExcha.txBuffer[3]:= 16#0C;
				VAR_CommandWriter.fbClientDataExcha.txBuffer[4]:= VAR_CommandWriter.fbClientDataExcha.txBuffer[2] +
															VAR_CommandWriter.fbClientDataExcha.txBuffer[3];
				VAR_CommandWriter.fbClientDataExcha.nbTransmittedChar := 5;
				VAR_CommandWriter.fbClientDataExcha.nbExpectedChar := 6;
			4:
				(*Crystal Switch - R14*)
				VAR_CommandWriter.fbClientDataExcha.txBuffer[0]:=16#02;
				VAR_CommandWriter.fbClientDataExcha.txBuffer[1]:=16#00;
				VAR_CommandWriter.fbClientDataExcha.txBuffer[2]:= F_ToASC('R');
				VAR_CommandWriter.fbClientDataExcha.txBuffer[3]:= 16#0E;
				VAR_CommandWriter.fbClientDataExcha.txBuffer[4]:= VAR_CommandWriter.fbClientDataExcha.txBuffer[2] +
															VAR_CommandWriter.fbClientDataExcha.txBuffer[3];
				VAR_CommandWriter.fbClientDataExcha.nbTransmittedChar := 5;
				VAR_CommandWriter.fbClientDataExcha.nbExpectedChar := 6;
			END_CASE

			VAR_CommandWriter.fbClientDataExcha(
								hSocket 		:= VAR_CommandWriter.hSocket,
								bExecute 	:= TRUE,
								PRM_RECEIVE_POLLING_TIME:= T#1s, (*temporisation de polling de réception*)
								PRM_RECEIVE_TIMEOUT	:= T#10s);	(*temporisation de timeout de communication*)
			VAR_CommandWriter.eStep := CLIENT_STATE_DATAEXCHA_WAIT;
		END_IF

	CLIENT_STATE_DATAEXCHA_WAIT:	(*Etape 4 - Attente de la fin de l'échange*)
		VAR_CommandWriter.fbClientDataExcha( bExecute := FALSE );
		IF NOT VAR_CommandWriter.fbClientDataExcha.bBusy THEN
			IF NOT VAR_CommandWriter.fbClientDataExcha.bError THEN
				VAR_CommandWriter.eStep 		:= CLIENT_STATE_DATA_ANALYSE;
			ELSE
				(* possible errors are logged inside of fbClientDataExcha function block *)
				VAR_CommandWriter.nStepInError := 4;
				VAR_CommandWriter.nErrId := 	VAR_CommandWriter.fbClientDataExcha.nErrId;	(*n° d'erreur hérité de la fonction Fb_clientDataExchange*)
				VAR_CommandWriter.ErrDescription :=	CONCAT(
												CONCAT(VAR_CommandWriter.fbClientDataExcha.ErrDescription, ' '),
												CONCAT(' -Trame: ',UDINT_TO_STRING(VAR_CommandWriter.nRequest))
												);
				VAR_CommandWriter.eStep :=	CLIENT_STATE_ERROR;
			END_IF
		END_IF
	CLIENT_STATE_DATA_ANALYSE:	(*Etape 5 - Analyse des données reçues*)
		(*si retour d'une trame signalant une erreur*)
		IF (VAR_CommandWriter.fbClientDataExcha.rxBuffer[2] = 16#80) THEN
				VAR_CommandWriter.nStepInError := 5;
				VAR_CommandWriter.nErrId :=  1;
				VAR_CommandWriter.ErrDescription := CONCAT(
								CONCAT( 'PACKET ERROR : ',F_ToCHR( VAR_CommandWriter.fbClientDataExcha.RxBuffer[6])),
								CONCAT(' -Trame: ',UDINT_TO_STRING(VAR_CommandWriter.nRequest))
								);
				VAR_CommandWriter.eStep :=	CLIENT_STATE_ERROR;
		ELSE
			(*Actualisation des état ok sur les actions + on refait tomber les commandes*)
			CASE VAR_CommandWriter.nRequest OF
				0:
					STATE_START_OK := TRUE;
					VAR_START := FALSE;
				1:
					STATE_STOP_OK := TRUE;
					VAR_STOP := FALSE;
				2:
					STATE_RESET_OK :=TRUE;
					VAR_RESET	:= FALSE;
				3:
					STATE_RAZ_THICK_OK :=TRUE;
					VAR_RAZ_THICK	:= FALSE;
				4:
					STATE_SWITCH_XTAL_OK:=TRUE;
					VAR_SWITCH_CRYSTAL := FALSE;
			END_CASE;
			(*réactualisation du n° de trame de commande à envoyer en fonction des demandes d'envoi active et de ce qui a déjà été
			transmis*)
			IF (VAR_CommandWriter.nRequest <1 AND VAR_STOP) THEN
				VAR_CommandWriter.nRequest :=1;
			ELSIF (VAR_CommandWriter.nRequest <2 AND VAR_RESET) THEN
				VAR_CommandWriter.nRequest :=2;
			ELSIF (VAR_CommandWriter.nRequest <3 AND VAR_RAZ_THICK) THEN
				VAR_CommandWriter.nRequest :=3;
			ELSIF (VAR_CommandWriter.nRequest <4 AND VAR_SWITCH_CRYSTAL) THEN
				VAR_CommandWriter.nRequest :=4;
			ELSE
				VAR_CommandWriter.nRequest := 0;
				STATE_ACTION_OK := TRUE;
			END_IF
			VAR_CommandWriter.eStep :=	CLIENT_STATE_IDLE;
		END_IF

	CLIENT_STATE_CLOSE_START:	(*Etape 6 - déclenchement fermeture du port*)
		VAR_CommandWriter.fbClose( bExecute := FALSE );
		VAR_CommandWriter.fbClose(
				hSocket:= VAR_CommandWriter.hSocket,
				bExecute:= TRUE );
		VAR_CommandWriter.eStep := CLIENT_STATE_CLOSE_WAIT;

	CLIENT_STATE_CLOSE_WAIT: (*Etape 7 - attente de la fermeture du port*)
		VAR_CommandWriter.fbClose( bExecute := FALSE );
		IF NOT VAR_CommandWriter.fbClose.bBusy THEN
			VAR_CommandWriter.bConnected := FALSE;
			MEMSET( ADR(hSocket), 0, SIZEOF(hSocket));
			IF VAR_CommandWriter.fbClose.bError THEN
				VAR_CommandWriter.nErrId := VAR_CommandWriter.fbClose.nErrId;
				VAR_CommandWriter.nStepInError := 7;
				VAR_CommandWriter.ErrDescription := CONCAT('FbClose Error : ', UDINT_TO_STRING(VAR_CommandWriter.fbClose.nErrId));
				VAR_CommandWriter.eStep := CLIENT_STATE_ERROR;
			ELSE
				VAR_CommandWriter.bBusy := FALSE;
				VAR_CommandWriter.bError := FALSE;
				VAR_CommandWriter.nErrId := 0;
				VAR_CommandWriter.eStep := CLIENT_STATE_IDLE;
			END_IF
		END_IF

	CLIENT_STATE_ERROR: (* Etape 8 : Error step *)
		VAR_CommandWriter.bError := TRUE;
		IF VAR_CommandWriter.bConnected THEN
			VAR_CommandWriter.eStep := CLIENT_STATE_CLOSE_START;
		ELSE
			VAR_CommandWriter.bBusy := FALSE;
			//IF DEF_COM_COMMAND.AR_DEF THEN
				VAR_CommandWriter.eStep := CLIENT_STATE_IDLE;
			//END_IF
		END_IF
END_CASE
END_ACTION

ACTION COM_PARAM:
CASE VAR_ParameterWriter.eStep OF
	CLIENT_STATE_IDLE:		(*Etape 0 - sequence d'échange à l'arrêt*)
		(*si autorisé ou exclusif si connecté*)
		IF VAR_ParameterWriter.bEnable XOR VAR_ParameterWriter.bConnected THEN
			VAR_ParameterWriter.bBusy := TRUE;
			VAR_ParameterWriter.bError := FALSE;
			VAR_ParameterWriter.nErrid := 0;
			IF VAR_ParameterWriter.bEnable THEN
				VAR_ParameterWriter.fbConnectTON( IN := FALSE );
				VAR_ParameterWriter.eStep := CLIENT_STATE_CONNECT_START;
			ELSE
				VAR_ParameterWriter.eStep := CLIENT_STATE_CLOSE_START;
			END_IF
		ELSIF VAR_ParameterWriter.bConnected THEN
			VAR_ParameterWriter.fbDataExchaTON( IN := FALSE );
			VAR_ParameterWriter.eStep := CLIENT_STATE_DATAEXCHA_START;
		ELSE
			VAR_ParameterWriter.bBusy := FALSE;
		END_IF

	CLIENT_STATE_CONNECT_START: (*Etape 1 - connexion au port*)
		(*temporisation de reconnexion*)
		VAR_ParameterWriter.fbConnectTON( IN := TRUE, PT := VAR_ParameterWriter.connectTime);
		(*si tempo de reconnexion ok*)
		IF VAR_ParameterWriter.fbConnectTON.Q THEN
			VAR_ParameterWriter.fbConnectTON( IN := FALSE );
			VAR_ParameterWriter.fbConnect(  bExecute := FALSE  );
			VAR_ParameterWriter.fbConnect(
						sRemoteHost		:= CONF_sRemoteHost,
						nRemotePort		:= CONF_nRemotePort,
						 sSrvNetId		:= '',
						bExecute		:= TRUE );
			VAR_ParameterWriter.eStep := CLIENT_STATE_CONNECT_WAIT;
			VAR_ParameterWriter.nRequest := 0; (*reinitalisation du n° de requete à 0*)
			VAR_ParameterWriter.Compteur_connection := VAR_ParameterWriter.Compteur_connection + 1;
		END_IF

	CLIENT_STATE_CONNECT_WAIT:	(*Etape 2 - attente connexion ok*)
		VAR_ParameterWriter.fbConnect( bExecute := FALSE );
		IF NOT VAR_ParameterWriter.fbConnect.bBusy THEN
			IF NOT VAR_ParameterWriter.fbConnect.bError THEN
				VAR_ParameterWriter.bConnected 	:= TRUE;
				VAR_ParameterWriter.hSocket 	:= VAR_ParameterWriter.fbConnect.hSocket;
				VAR_ParameterWriter.eStep 		:= CLIENT_STATE_IDLE;
				Def_connect_com_parameters := FALSE;
			ELSE
				VAR_ParameterWriter.nErrId := VAR_ParameterWriter.fbConnect.nErrId;
				VAR_ParameterWriter.nStepInError  := 2;
				VAR_ParameterWriter.ErrDescription := CONCAT('FbConnect Error : ', UDINT_TO_STRING(VAR_ParameterWriter.fbConnect.nErrId));
				VAR_ParameterWriter.eStep := CLIENT_STATE_ERROR;
				Def_connect_com_parameters := TRUE;
			END_IF
		END_IF

	CLIENT_STATE_DATAEXCHA_START:	(*Etape 3 - lancement des échanges*)
		VAR_ParameterWriter.fbDataExchaTON( IN := TRUE, PT := VAR_ParameterWriter.ExchangeCycleTime );
		IF VAR_ParameterWriter.fbDataExchaTON.Q THEN
			VAR_ParameterWriter.fbDataExchaTON( IN := FALSE );
			VAR_ParameterWriter.fbClientDataExcha( bExecute := FALSE );


			CASE VAR_ParameterWriter.nRequest OF

						0:	(*Rise Time 1*)
							VAR_ParameterWriter.fbClientDataExcha.txBuffer[0]:=16#08;
							VAR_ParameterWriter.fbClientDataExcha.txBuffer[1]:=16#00;
							VAR_ParameterWriter.fbClientDataExcha.txBuffer[2]:= F_ToASC('U');
							VAR_ParameterWriter.fbClientDataExcha.txBuffer[3]:= F_ToASC('F');
							VAR_ParameterWriter.fbClientDataExcha.txBuffer[4]:= 16#00;
							VAR_ParameterWriter.fbClientDataExcha.txBuffer[5]:= 16#01;
							TEMP_DWORD := INT_TO_DWORD(I_Rise_Time_1);
							MEMCPY(ADR(VAR_ParameterWriter.fbClientDataExcha.txBuffer[6]),ADR(TEMP_DWORD),4);
							VAR_ParameterWriter.fbClientDataExcha.txBuffer[10] := VAR_ParameterWriter.fbClientDataExcha.txBuffer[2] +
												VAR_ParameterWriter.fbClientDataExcha.txBuffer[3] +
												VAR_ParameterWriter.fbClientDataExcha.txBuffer[4] +
												VAR_ParameterWriter.fbClientDataExcha.txBuffer[5] +
												VAR_ParameterWriter.fbClientDataExcha.txBuffer[6] +
												VAR_ParameterWriter.fbClientDataExcha.txBuffer[7] +
												VAR_ParameterWriter.fbClientDataExcha.txBuffer[8] +
												VAR_ParameterWriter.fbClientDataExcha.txBuffer[9];
							VAR_ParameterWriter.fbClientDataExcha.nbTransmittedChar := 11;
							VAR_ParameterWriter.fbClientDataExcha.nbExpectedChar := 6;


						1:	(*Soak Power 1*)
							VAR_ParameterWriter.fbClientDataExcha.txBuffer[0]:=16#08;
							VAR_ParameterWriter.fbClientDataExcha.txBuffer[1]:=16#00;
							VAR_ParameterWriter.fbClientDataExcha.txBuffer[2]:= F_ToASC('U');
							VAR_ParameterWriter.fbClientDataExcha.txBuffer[3]:= F_ToASC('F');
							VAR_ParameterWriter.fbClientDataExcha.txBuffer[4]:= 16#01;
							VAR_ParameterWriter.fbClientDataExcha.txBuffer[5]:= 16#01;
							MEMCPY(ADR(VAR_ParameterWriter.fbClientDataExcha.txBuffer[6]),ADR(I_Soak_Power_1),4);
							VAR_ParameterWriter.fbClientDataExcha.txBuffer[10] := VAR_ParameterWriter.fbClientDataExcha.txBuffer[2] +
												VAR_ParameterWriter.fbClientDataExcha.txBuffer[3] +
												VAR_ParameterWriter.fbClientDataExcha.txBuffer[4] +
												VAR_ParameterWriter.fbClientDataExcha.txBuffer[5] +
												VAR_ParameterWriter.fbClientDataExcha.txBuffer[6] +
												VAR_ParameterWriter.fbClientDataExcha.txBuffer[7] +
												VAR_ParameterWriter.fbClientDataExcha.txBuffer[8] +
												VAR_ParameterWriter.fbClientDataExcha.txBuffer[9];
							VAR_ParameterWriter.fbClientDataExcha.nbTransmittedChar := 11;
							VAR_ParameterWriter.fbClientDataExcha.nbExpectedChar := 6;


						2:	(*Soak Time 1*)
							VAR_ParameterWriter.fbClientDataExcha.txBuffer[0]:=16#08;
							VAR_ParameterWriter.fbClientDataExcha.txBuffer[1]:=16#00;
							VAR_ParameterWriter.fbClientDataExcha.txBuffer[2]:= F_ToASC('U');
							VAR_ParameterWriter.fbClientDataExcha.txBuffer[3]:= F_ToASC('F');
							VAR_ParameterWriter.fbClientDataExcha.txBuffer[4]:= 16#02;
							VAR_ParameterWriter.fbClientDataExcha.txBuffer[5]:= 16#01;
							TEMP_DWORD := INT_TO_DWORD(I_Soak_Time_1);
							MEMCPY(ADR(VAR_ParameterWriter.fbClientDataExcha.txBuffer[6]),ADR(TEMP_DWORD),4);
							VAR_ParameterWriter.fbClientDataExcha.txBuffer[10] := VAR_ParameterWriter.fbClientDataExcha.txBuffer[2] +
												VAR_ParameterWriter.fbClientDataExcha.txBuffer[3] +
												VAR_ParameterWriter.fbClientDataExcha.txBuffer[4] +
												VAR_ParameterWriter.fbClientDataExcha.txBuffer[5] +
												VAR_ParameterWriter.fbClientDataExcha.txBuffer[6] +
												VAR_ParameterWriter.fbClientDataExcha.txBuffer[7] +
												VAR_ParameterWriter.fbClientDataExcha.txBuffer[8] +
												VAR_ParameterWriter.fbClientDataExcha.txBuffer[9];
							VAR_ParameterWriter.fbClientDataExcha.nbTransmittedChar := 11;
							VAR_ParameterWriter.fbClientDataExcha.nbExpectedChar := 6;


						3:	(*Rise Time 2*)
							VAR_ParameterWriter.fbClientDataExcha.TxBuffer[0]:=16#08;
							VAR_ParameterWriter.fbClientDataExcha.txBuffer[1]:=16#00;
							VAR_ParameterWriter.fbClientDataExcha.txBuffer[2]:= F_ToASC('U');
							VAR_ParameterWriter.fbClientDataExcha.txBuffer[3]:= F_ToASC('F');
							VAR_ParameterWriter.fbClientDataExcha.txBuffer[4]:= 16#03;
							VAR_ParameterWriter.fbClientDataExcha.txBuffer[5]:= 16#01;
							TEMP_DWORD := INT_TO_DWORD(I_Rise_Time_2);
							MEMCPY(ADR(VAR_ParameterWriter.fbClientDataExcha.txBuffer[6]),ADR(TEMP_DWORD),4);
							VAR_ParameterWriter.fbClientDataExcha.txBuffer[10] := VAR_ParameterWriter.fbClientDataExcha.txBuffer[2] +
												VAR_ParameterWriter.fbClientDataExcha.txBuffer[3] +
												VAR_ParameterWriter.fbClientDataExcha.txBuffer[4] +
												VAR_ParameterWriter.fbClientDataExcha.txBuffer[5] +
												VAR_ParameterWriter.fbClientDataExcha.txBuffer[6] +
												VAR_ParameterWriter.fbClientDataExcha.txBuffer[7] +
												VAR_ParameterWriter.fbClientDataExcha.txBuffer[8] +
												VAR_ParameterWriter.fbClientDataExcha.txBuffer[9];
							VAR_ParameterWriter.fbClientDataExcha.nbTransmittedChar := 11;
							VAR_ParameterWriter.fbClientDataExcha.nbExpectedChar := 6;


						4:	(*Soak Power 2*)
							VAR_ParameterWriter.fbClientDataExcha.txBuffer[0]:=16#08;
							VAR_ParameterWriter.fbClientDataExcha.txBuffer[1]:=16#00;
							VAR_ParameterWriter.fbClientDataExcha.txBuffer[2]:= F_ToASC('U');
							VAR_ParameterWriter.fbClientDataExcha.txBuffer[3]:= F_ToASC('F');
							VAR_ParameterWriter.fbClientDataExcha.txBuffer[4]:= 16#04;
							VAR_ParameterWriter.fbClientDataExcha.txBuffer[5]:= 16#01;
							MEMCPY(ADR(VAR_ParameterWriter.fbClientDataExcha.txBuffer[6]),ADR(I_Soak_Power_2),4);
							VAR_ParameterWriter.fbClientDataExcha.txBuffer[10] := VAR_ParameterWriter.fbClientDataExcha.txBuffer[2] +
												VAR_ParameterWriter.fbClientDataExcha.txBuffer[3] +
												VAR_ParameterWriter.fbClientDataExcha.txBuffer[4] +
												VAR_ParameterWriter.fbClientDataExcha.txBuffer[5] +
												VAR_ParameterWriter.fbClientDataExcha.txBuffer[6] +
												VAR_ParameterWriter.fbClientDataExcha.txBuffer[7] +
												VAR_ParameterWriter.fbClientDataExcha.txBuffer[8] +
												VAR_ParameterWriter.fbClientDataExcha.txBuffer[9];
							VAR_ParameterWriter.fbClientDataExcha.nbTransmittedChar := 11;
							VAR_ParameterWriter.fbClientDataExcha.nbExpectedChar := 6;


						5:	(*Soak Time 2*)
							VAR_ParameterWriter.fbClientDataExcha.txBuffer[0]:=16#08;
							VAR_ParameterWriter.fbClientDataExcha.txBuffer[1]:=16#00;
							VAR_ParameterWriter.fbClientDataExcha.txBuffer[2]:= F_ToASC('U');
							VAR_ParameterWriter.fbClientDataExcha.txBuffer[3]:= F_ToASC('F');
							VAR_ParameterWriter.fbClientDataExcha.txBuffer[4]:= 16#05;
							VAR_ParameterWriter.fbClientDataExcha.txBuffer[5]:= 16#01;
							TEMP_DWORD := INT_TO_DWORD(I_Soak_Time_2);
							MEMCPY(ADR(VAR_ParameterWriter.fbClientDataExcha.txBuffer[6]),ADR(TEMP_DWORD),4);
							VAR_ParameterWriter.fbClientDataExcha.txBuffer[10] := VAR_ParameterWriter.fbClientDataExcha.txBuffer[2] +
												VAR_ParameterWriter.fbClientDataExcha.txBuffer[3] +
												VAR_ParameterWriter.fbClientDataExcha.txBuffer[4] +
												VAR_ParameterWriter.fbClientDataExcha.txBuffer[5] +
												VAR_ParameterWriter.fbClientDataExcha.txBuffer[6] +
												VAR_ParameterWriter.fbClientDataExcha.txBuffer[7] +
												VAR_ParameterWriter.fbClientDataExcha.txBuffer[8] +
												VAR_ParameterWriter.fbClientDataExcha.txBuffer[9];
							VAR_ParameterWriter.fbClientDataExcha.nbTransmittedChar := 11;
							VAR_ParameterWriter.fbClientDataExcha.nbExpectedChar := 6;


						6:	(*Idle Ramp*)
							VAR_ParameterWriter.fbClientDataExcha.txBuffer[0]:=16#08;
							VAR_ParameterWriter.fbClientDataExcha.txBuffer[1]:=16#00;
							VAR_ParameterWriter.fbClientDataExcha.txBuffer[2]:= F_ToASC('U');
							VAR_ParameterWriter.fbClientDataExcha.txBuffer[3]:= F_ToASC('F');
							VAR_ParameterWriter.fbClientDataExcha.txBuffer[4]:= 16#06;
							VAR_ParameterWriter.fbClientDataExcha.txBuffer[5]:= 16#01;
							TEMP_DWORD :=INT_TO_DWORD(I_Idle_Ramp);
							MEMCPY(ADR(VAR_ParameterWriter.fbClientDataExcha.txBuffer[6]),ADR(TEMP_DWORD),4);
							VAR_ParameterWriter.fbClientDataExcha.txBuffer[10] := VAR_ParameterWriter.fbClientDataExcha.txBuffer[2] +
												VAR_ParameterWriter.fbClientDataExcha.txBuffer[3] +
												VAR_ParameterWriter.fbClientDataExcha.txBuffer[4] +
												VAR_ParameterWriter.fbClientDataExcha.txBuffer[5] +
												VAR_ParameterWriter.fbClientDataExcha.txBuffer[6] +
												VAR_ParameterWriter.fbClientDataExcha.txBuffer[7] +
												VAR_ParameterWriter.fbClientDataExcha.txBuffer[8] +
												VAR_ParameterWriter.fbClientDataExcha.txBuffer[9];
							VAR_ParameterWriter.fbClientDataExcha.nbTransmittedChar := 11;
							VAR_ParameterWriter.fbClientDataExcha.nbExpectedChar := 6;


						7:	(*Idle Power*)
							VAR_ParameterWriter.fbClientDataExcha.txBuffer[0]:=16#08;
							VAR_ParameterWriter.fbClientDataExcha.txBuffer[1]:=16#00;
							VAR_ParameterWriter.fbClientDataExcha.txBuffer[2]:= F_ToASC('U');
							VAR_ParameterWriter.fbClientDataExcha.txBuffer[3]:= F_ToASC('F');
							VAR_ParameterWriter.fbClientDataExcha.txBuffer[4]:= 16#07;
							VAR_ParameterWriter.fbClientDataExcha.txBuffer[5]:= 16#01;
							MEMCPY(ADR(VAR_ParameterWriter.fbClientDataExcha.txBuffer[6]),ADR(I_Idle_Power),4);
							VAR_ParameterWriter.fbClientDataExcha.txBuffer[10] := VAR_ParameterWriter.fbClientDataExcha.txBuffer[2] +
												VAR_ParameterWriter.fbClientDataExcha.txBuffer[3] +
												VAR_ParameterWriter.fbClientDataExcha.txBuffer[4] +
												VAR_ParameterWriter.fbClientDataExcha.txBuffer[5] +
												VAR_ParameterWriter.fbClientDataExcha.txBuffer[6] +
												VAR_ParameterWriter.fbClientDataExcha.txBuffer[7] +
												VAR_ParameterWriter.fbClientDataExcha.txBuffer[8] +
												VAR_ParameterWriter.fbClientDataExcha.txBuffer[9];
							VAR_ParameterWriter.fbClientDataExcha.nbTransmittedChar := 11;
							VAR_ParameterWriter.fbClientDataExcha.nbExpectedChar := 6;


						8:	(*Consigne de Vitesse d'évaporation*)
							VAR_ParameterWriter.fbClientDataExcha.txBuffer[0]:=16#08;
							VAR_ParameterWriter.fbClientDataExcha.txBuffer[1]:=16#00;
							VAR_ParameterWriter.fbClientDataExcha.txBuffer[2]:= F_ToASC('U');
							VAR_ParameterWriter.fbClientDataExcha.txBuffer[3]:= F_ToASC('F');
							VAR_ParameterWriter.fbClientDataExcha.txBuffer[4]:= 16#08;
							VAR_ParameterWriter.fbClientDataExcha.txBuffer[5]:= 16#01;
							MEMCPY(ADR(VAR_ParameterWriter.fbClientDataExcha.txBuffer[6]),ADR(I_Deposition_Rate),4);
							VAR_ParameterWriter.fbClientDataExcha.txBuffer[10] := VAR_ParameterWriter.fbClientDataExcha.txBuffer[2] +
												VAR_ParameterWriter.fbClientDataExcha.txBuffer[3] +
												VAR_ParameterWriter.fbClientDataExcha.txBuffer[4] +
												VAR_ParameterWriter.fbClientDataExcha.txBuffer[5] +
												VAR_ParameterWriter.fbClientDataExcha.txBuffer[6] +
												VAR_ParameterWriter.fbClientDataExcha.txBuffer[7] +
												VAR_ParameterWriter.fbClientDataExcha.txBuffer[8] +
												VAR_ParameterWriter.fbClientDataExcha.txBuffer[9];
							VAR_ParameterWriter.fbClientDataExcha.nbTransmittedChar := 11;
							VAR_ParameterWriter.fbClientDataExcha.nbExpectedChar := 6;



						9:	(*Consigne d'épaisseur*)
							VAR_ParameterWriter.fbClientDataExcha.txBuffer[0]:=16#08;
							VAR_ParameterWriter.fbClientDataExcha.txBuffer[1]:=16#00;
							VAR_ParameterWriter.fbClientDataExcha.txBuffer[2]:= F_ToASC('U');
							VAR_ParameterWriter.fbClientDataExcha.txBuffer[3]:= F_ToASC('F');
							VAR_ParameterWriter.fbClientDataExcha.txBuffer[4]:= 16#09;
							VAR_ParameterWriter.fbClientDataExcha.txBuffer[5]:= 16#01;
							MEMCPY(ADR(VAR_ParameterWriter.fbClientDataExcha.txBuffer[6]),ADR(I_Final_thickness),4);
							VAR_ParameterWriter.fbClientDataExcha.txBuffer[10] := VAR_ParameterWriter.fbClientDataExcha.txBuffer[2] +
												VAR_ParameterWriter.fbClientDataExcha.txBuffer[3] +
												VAR_ParameterWriter.fbClientDataExcha.txBuffer[4] +
												VAR_ParameterWriter.fbClientDataExcha.txBuffer[5] +
												VAR_ParameterWriter.fbClientDataExcha.txBuffer[6] +
												VAR_ParameterWriter.fbClientDataExcha.txBuffer[7] +
												VAR_ParameterWriter.fbClientDataExcha.txBuffer[8] +
												VAR_ParameterWriter.fbClientDataExcha.txBuffer[9];
							VAR_ParameterWriter.fbClientDataExcha.nbTransmittedChar := 11;
							VAR_ParameterWriter.fbClientDataExcha.nbExpectedChar := 6;


